	FUNCTION FC 817  : VOID
	TITLE =MAL1S017 Section control: LINE 1 SEC 17 GERM 1
	//COPYRIGHT:    (C) 2009 BY  BUHLER AG
	//                           CH-9240 UZWIL  SWITZERLAND
	//
	//PRODUCT:      WinCoS_BIW01_09
	//
	//TITLE:        LINE 1 SEC 17 GERM 1
	//                 Section control
	//
	//--------------------------------------------------------------------------------
	//
	//IDENT:        AUTHOR:             DEPT:                              DATE:
	//
	//P01_FC817.1.0 K.Renz              CSB41                              13.Jan.2010
	//              1st Release
	//
	//--------------------------------------------------------------------------------
	//
	//PURPOSE:
	//
	//REFERENCES : GCSOSMAN
	//
	//--------------------------------------------------------------------------------
	//
	//
	AUTHOR  : KR
	FAMILY  : USW
	VERSION : 9.9
	//0000 to 0999: Main Functions
	//              0 =Main Function Cylic
	//              1 =Main Function Coldstart/Newstart
	//              2 =Main Function Warm Start

	VAR_INPUT
	  InCode : INT ;
	END_VAR

	VAR_TEMP
	tmpStartNext : BOOL ;	//Condition to Start next element
	tmpFlagFault : BOOL ;	//Flag mechanical fault
	tmpEnableFeed : BOOL ;
	tmpStartScale : BOOL ;
	tmpStartLiqScale : BOOL ; //Enable to Start Lipquid Scale
	tmpSndBin: Int ;
	tmpRcvBin: Int ;
	tmpBool : BOOL ;
	tmpByte : BYTE ;
	tmpWord : WORD ;
	tmpDWord : DWORD ;
	tmpInt : INT ;
	tmpRET : INT ;
	tmpDInt : DINT ;
	tmpCyclusTime : DINT ;
	tmpWetSteep : BOOL ;
	END_VAR

	BEGIN

	NETWORK
	TITLE =
	//=================================================
	//=================================================
	//S T A R T   M A I N   F U N C T I O N
	//=================================================
	//=================================================
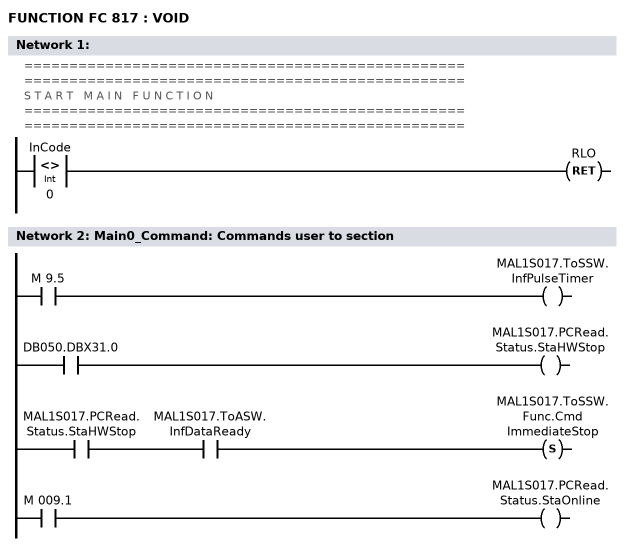
	      L InCode;
	      L 0;
	      <>I;
	      BEB;

	NETWORK
	TITLE =Main0_Command: Commands user to section
	      NOP   0;
	//-Tick 1 second---
		U     M 9.5;
		=     MAL1S017.ToSSW.InfPulseTimer;
	//-Hardware stop---
		U     DB050.DBX31.0 ;
		=     MAL1S017.PCRead.Status.StaHWStop;
		U   MAL1S017.PCRead.Status.StaHWStop;
		U   MAL1S017.ToASW.InfDataReady;
		S     MAL1S017.ToSSW.Func.CmdImmediateStop;
	//-Online---
		U     M 009.1 ;
		=     MAL1S017.PCRead.Status.StaOnline;
	NETWORK
	TITLE =ASW_UC: User commands to section
	NOP 0;
	//-Additional user commands---
	//-GP standard commands---
	      AUF   "MAL1S017" ;
	      L     L#0 ;                           // Enter the differenz of the target weight and prestop weight
	      T    "MAL1S017".VarTemp.InOutValue3;  // Prestop weight
	      CALL FC   120 (
	           InCode                   := 2001);// Section function: Standard section commands

	//-Condition CmdSequenzStop---
	      U     MAL1S017.ToSSW.Func.CmdSequenzStop;
	//      S     "MAL1S017".ToSSW.Func.CmdSequenzStop
	      R     MAL1S017.ToSSW.Func.CmdSequenzStop;
	//-Extended section commands---
	      AUF   "MAL1S017";
	      CALL "STD_LineSecStdSub" (
	           InCode                   := 2002);// Section function: Extended section commands
	//-Status from pulse commands---
	      CLR;
	      =     DB817.DBX  157.0;
	      =     DB817.DBX  157.1;
	      =     DB817.DBX  157.2;
	      =     DB817.DBX  157.3;
	      =     DB817.DBX  157.4;
	      =     DB817.DBX  157.5;
	      =     DB817.DBX  157.6;
	      =     DB817.DBX  157.7;
	//
	NETWORK
	TITLE =Main0_Dest: Destination
	NETWORK
	TITLE =Main0_Next: Ready for next batch

		ON    MAL1S017.ToASW.InfDataReady;
		=     MAL1S017.ToSSW.InfReadyForNewBatch;
	NETWORK
	TITLE =Main0_Control: Control section
	      NOP   0;
	//-Process commands from PCS---
		AUF   "MAL1S017" ;
		CALL FC    60 (// Methode O_Section
		CODE                     := 7);
	//-Process commands from user---
		AUF   "MAL1S017" ;
		CALL FC    60 (// Methode Control
		CODE                     := 0);
	//-Process section step---
		AUF   "MAL1S017" ;
		CALL FC    60 (// Methode Step_execute
		CODE                     := 2);
		AUF   "MAL1S017" ;
		CALL FC    60 (// Methode Step_transition
		CODE                     := 3);
	//-Process section state---
		AUF   "MAL1S017" ;
		CALL FC    60 (// Methode State
		CODE                     := 4);

	NETWORK
	TITLE =Main0_Init: Init
		UN    MAL1S017.ToASW.Transition.ToWait;
		UN    MAL1S017.ToASW.CmdNewBatch;
		SPB   in00;
	//-User initialization---
		AUF   "MAL1S017" ;
	//
	//-Section function: Init ---
		AUF   "MAL1S017" ;
	      CALL FC   120 (
	           InCode                   := 2003);// Section function: Init
	//
	//-Group interface---
	//
	//-Initialise bin objects---
	//
	//-Emptying job---
	      U    MAL1S017.JobAc.StaBatch.StaEmptyingBatch;
	      S     MAL1S017.PCRead.Status.StaLoaded;
	//
	//-Error Batch---
	//
	in00:	NOP   0;

	NETWORK
	TITLE =ASW_VB: Various functions before bin control
	      NOP   0;
	//
	//-Update staSameSndRcv in sender binlist---
	NETWORK
	TITLE =Main0_GrNRS: Not Relevant for started / Fault
		NOP 0;
	      SET;
	      =     "MAL1S017".Gr.ParNotRelForStarted[103];
	      =     "MAL1S017".Gr.ParNotRelForStarted[105];
	      =     "MAL1S017".Gr.ParNotRelForStarted[106];
	      =     "MAL1S017".Gr.ParNotRelForStarted[107];
	      =     "MAL1S017".Gr.ParNotRelForStarted[108];
	      =     "MAL1S017".Gr.ParNotRelForStarted[109];
	      =     "MAL1S017".Gr.ParNotRelForStarted[112];
	      =     "MAL1S017".Gr.ParNotRelForFault[103];
	      =     "MAL1S017".Gr.ParNotRelForFault[105];
	      =     "MAL1S017".Gr.ParNotRelForFault[106];
	      =     "MAL1S017".Gr.ParNotRelForFault[107];
	      =     "MAL1S017".Gr.ParNotRelForFault[108];
	      =     "MAL1S017".Gr.ParNotRelForFault[109];
	      =     "MAL1S017".Gr.ParNotRelForFault[112];
	NETWORK
	TITLE =Main0_GrSelection: Group selection
	// List of the used objects in the section
	// ==========================
	// G005G       GENERAL ELEMENTS GERM 1
	// G091F       BELT CONVEYOR 4100 GERM 1-4
	// G092F       BELT CONVEYOR 4200 GERM 5-8
	// G093M       BELT CONVEYOR 4300 GERM
	// G094M       BELT CONVEYOR 4400 GERM
	// G095M       BELT CONVEYOR 4500 GERM
	// G097M       LIFTING DEVICE GERM 1
	// G098M       COUPLING DEVICE TURNER GERM 1
	// G099M       COUPLING DEVICE WALL GERM 1
	// G100M       TRAVELLING DRIVE GERM 1
	// G101M       HORIZONTAL AND LIFTING SCREW GERM 1
	// G102M       LOCAL COMMAND BUTTON / LAMPS GERM 1
	// G103M       TEMPERATURE MES. GERM 1
	// G104M       TURNING SCREWS GERM 1
	// G105M       FAN AND VALVE SRAY AIR GERM 1
	// G106M       FRESH AIR LOUVER GERM 1
	// G107M       EXHAUST AIR LOUVER GERM 1
	// G108M       PRODUCT MOISTERING  GERM 1
	// G109M       HP CLEANING GERM 1
	// G110M       INLET SLIDE GERM 1
	// G111M       LOADING CONVEYOR 4600 GERM 1
	// G112M       COOLING / HEATING GERM 1
	// G113M       BELT CONVEYOR 7050 GERM 1 / 2
	//
	      NOP   0;
//-Condition for preselection---
		U     MAL1S017.ToASW.InfDataReady;
		SPB   GS01;
//-Deselect groups ---
		CALL FB     9 , "GCS7_GrCtrlDBTmp" (// GrCtr.Methode Deselect
		     Code  := 3,
		     Sec   := "MAL1S017".Gr);
		SPA   GS02;
//-Select groups ---
	GS01:	NOP 0;
	//-Prepare for preselection ---
		CALL FB     9 , "GCS7_GrCtrlDBTmp" (// GrCtr.Methode Init Preselection
		     Code  := 1,
		     Sec   := "MAL1S017".Gr);
	//
	//
	//-Prestart used groups --
		U     M     50.0;
		=     M     50.0;

	//-Preselect used groups --
		U     M     50.0;
		=     M     50.0;
		S   MAL1S017.Gr.InPreselect[5];   //-->G005G GENERAL ELEMENTS GERM 1
		S   MAL1S017.Gr.InPreselect[91];   //-->G091F BELT CONVEYOR 4100 GERM 1-4
		S   MAL1S017.Gr.InPreselect[92];   //-->G092F BELT CONVEYOR 4200 GERM 5-8
		S   MAL1S017.Gr.InPreselect[93];   //-->G093M BELT CONVEYOR 4300 GERM
		S   MAL1S017.Gr.InPreselect[94];   //-->G094M BELT CONVEYOR 4400 GERM
		S   MAL1S017.Gr.InPreselect[95];   //-->G095M BELT CONVEYOR 4500 GERM
		S   MAL1S017.Gr.InPreselect[97];   //-->G097M LIFTING DEVICE GERM 1
		S   MAL1S017.Gr.InPreselect[98];   //-->G098M COUPLING DEVICE TURNER GERM 1
		S   MAL1S017.Gr.InPreselect[99];   //-->G099M COUPLING DEVICE WALL GERM 1
		S   MAL1S017.Gr.InPreselect[100];   //-->G100M TRAVELLING DRIVE GERM 1
		S   MAL1S017.Gr.InPreselect[101];   //-->G101M HORIZONTAL AND LIFTING SCREW GERM 1
		S   MAL1S017.Gr.InPreselect[102];   //-->G102M LOCAL COMMAND BUTTON / LAMPS GERM 1
		S   MAL1S017.Gr.InPreselect[103];   //-->G103M TEMPERATURE MES. GERM 1
		S   MAL1S017.Gr.InPreselect[104];   //-->G104M TURNING SCREWS GERM 1
		S   MAL1S017.Gr.InPreselect[105];   //-->G105M FAN AND VALVE SRAY AIR GERM 1
		S   MAL1S017.Gr.InPreselect[106];   //-->G106M FRESH AIR LOUVER GERM 1
		S   MAL1S017.Gr.InPreselect[107];   //-->G107M EXHAUST AIR LOUVER GERM 1
		S   MAL1S017.Gr.InPreselect[108];   //-->G108M PRODUCT MOISTERING  GERM 1
		S   MAL1S017.Gr.InPreselect[109];   //-->G109M HP CLEANING GERM 1
		S   MAL1S017.Gr.InPreselect[110];   //-->G110M INLET SLIDE GERM 1
		S   MAL1S017.Gr.InPreselect[111];   //-->G111M LOADING CONVEYOR 4600 GERM 1
		S   MAL1S017.Gr.InPreselect[112];   //-->G112M COOLING / HEATING GERM 1
		S   MAL1S017.Gr.InPreselect[113];   //-->G113M BELT CONVEYOR 7050 GERM 1 / 2
	      L     1;
	      L     "MAL1S017Par".StepAct.StepNumber;
	      UW;
	      ==I;  // step wetsteep
	      =    "MAL1S017Par".Par.FlagGen.WetStep;

	//
	//-Set CmdNewJob ---
	     U     MAL1S017.Gr.InPreselect[91];
	     UN    #GCS7_GrCtrlDB.OutOccupied[91];
	     S       G091F.CmdNewJob;
	     U     MAL1S017.Gr.InPreselect[92];
	     UN    #GCS7_GrCtrlDB.OutOccupied[92];
	     S       G092F.CmdNewJob;
	     U     MAL1S017.Gr.InPreselect[93];
	     UN    #GCS7_GrCtrlDB.OutOccupied[93];
	     S       G093M.CmdNewJob;
	     U     MAL1S017.Gr.InPreselect[94];
	     UN    #GCS7_GrCtrlDB.OutOccupied[94];
	     S       G094M.CmdNewJob;
	     U     MAL1S017.Gr.InPreselect[95];
	     UN    #GCS7_GrCtrlDB.OutOccupied[95];
	     S       G095M.CmdNewJob;
	     U     MAL1S017.Gr.InPreselect[97];
	     UN    #GCS7_GrCtrlDB.OutOccupied[97];
	     S       G097M.CmdNewJob;
	     U     MAL1S017.Gr.InPreselect[98];
	     UN    #GCS7_GrCtrlDB.OutOccupied[98];
	     S       G098M.CmdNewJob;
	     U     MAL1S017.Gr.InPreselect[99];
	     UN    #GCS7_GrCtrlDB.OutOccupied[99];
	     S       G099M.CmdNewJob;
	     U     MAL1S017.Gr.InPreselect[100];
	     UN    #GCS7_GrCtrlDB.OutOccupied[100];
	     S       G100M.CmdNewJob;
	     U     MAL1S017.Gr.InPreselect[101];
	     UN    #GCS7_GrCtrlDB.OutOccupied[101];
	     S       G101M.CmdNewJob;
	     U     MAL1S017.Gr.InPreselect[102];
	     UN    #GCS7_GrCtrlDB.OutOccupied[102];
	     S       G102M.CmdNewJob;
	     U     MAL1S017.Gr.InPreselect[103];
	     UN    #GCS7_GrCtrlDB.OutOccupied[103];
	     S       G103M.CmdNewJob;
	     U     MAL1S017.Gr.InPreselect[104];
	     UN    #GCS7_GrCtrlDB.OutOccupied[104];
	     S       G104M.CmdNewJob;
	     U     MAL1S017.Gr.InPreselect[105];
	     UN    #GCS7_GrCtrlDB.OutOccupied[105];
	     S       G105M.CmdNewJob;
	     U     MAL1S017.Gr.InPreselect[106];
	     UN    #GCS7_GrCtrlDB.OutOccupied[106];
	     S       G106M.CmdNewJob;
	     U     MAL1S017.Gr.InPreselect[107];
	     UN    #GCS7_GrCtrlDB.OutOccupied[107];
	     S       G107M.CmdNewJob;
	     U     MAL1S017.Gr.InPreselect[108];
	     UN    #GCS7_GrCtrlDB.OutOccupied[108];
	     S       G108M.CmdNewJob;
	     U     MAL1S017.Gr.InPreselect[109];
	     UN    #GCS7_GrCtrlDB.OutOccupied[109];
	     S       G109M.CmdNewJob;
	     U     MAL1S017.Gr.InPreselect[110];
	     UN    #GCS7_GrCtrlDB.OutOccupied[110];
	     S       G110M.CmdNewJob;
	     U     MAL1S017.Gr.InPreselect[111];
	     UN    #GCS7_GrCtrlDB.OutOccupied[111];
	     S       G111M.CmdNewJob;
	     U     MAL1S017.Gr.InPreselect[112];
	     UN    #GCS7_GrCtrlDB.OutOccupied[112];
	     S       G112M.CmdNewJob;
	     U     MAL1S017.Gr.InPreselect[113];
	     UN    #GCS7_GrCtrlDB.OutOccupied[113];
	     S       G113M.CmdNewJob;
	//
	//
	//-Test preselected groups ---
		CALL FB     9 , "GCS7_GrCtrlDBTmp" (// GrCtr.Methode Select
		     Code  := 2,
		     Sec   := "MAL1S017".Gr);
	//
	//-Way conflict if not available---
		CLR;
		S     MAL1S017.Gr.All.OutGrConflict;
	//
	//-Test occupied real and virtual groups---
	GS02:   NOP 0;
		U     MAL1S017.Gr.All.OutSelectionValid;
		UN    MAL1S017.Gr.All.OutGrIsLocked;
		=     MAL1S017.Gr.All.InOutASWSelectionOK;
	//
	//
	//----- Send data to selected groups =====
	GS3:	UN  MAL1S017.Gr.OutSelected[91]; //G091F
		SPB GS4;
		L     "MAL1".Para.ParLineNr;
		T     G091F.Gr.InLine;
	GS4:	UN  MAL1S017.Gr.OutSelected[92]; //G092F
		SPB GS5;
		L     "MAL1".Para.ParLineNr;
		T     G092F.Gr.InLine;
	GS5:	UN  MAL1S017.Gr.OutSelected[93]; //G093M
		SPB GS6;
		L     "MAL1".Para.ParLineNr;
		T     G093M.Gr.InLine;
	GS6:	UN  MAL1S017.Gr.OutSelected[94]; //G094M
		SPB GS7;
		L     "MAL1".Para.ParLineNr;
		T     G094M.Gr.InLine;
	GS7:	UN  MAL1S017.Gr.OutSelected[95]; //G095M
		SPB GS8;
		L     "MAL1".Para.ParLineNr;
		T     G095M.Gr.InLine;
	GS8:	UN  MAL1S017.Gr.OutSelected[97]; //G097M
		SPB GS9;
		L     "MAL1".Para.ParLineNr;
		T     G097M.Gr.InLine;
	GS9:	UN  MAL1S017.Gr.OutSelected[98]; //G098M
		SPB GS10;
		L     "MAL1".Para.ParLineNr;
		T     G098M.Gr.InLine;
	GS10:	UN  MAL1S017.Gr.OutSelected[99]; //G099M
		SPB GS11;
		L     "MAL1".Para.ParLineNr;
		T     G099M.Gr.InLine;
	GS11:	UN  MAL1S017.Gr.OutSelected[100]; //G100M
		SPB GS12;
		L     "MAL1".Para.ParLineNr;
		T     G100M.Gr.InLine;
	GS12:	UN  MAL1S017.Gr.OutSelected[101]; //G101M
		SPB GS13;
		L     "MAL1".Para.ParLineNr;
		T     G101M.Gr.InLine;
	GS13:	UN  MAL1S017.Gr.OutSelected[102]; //G102M
		SPB GS14;
		L     "MAL1".Para.ParLineNr;
		T     G102M.Gr.InLine;
	GS14:	UN  MAL1S017.Gr.OutSelected[103]; //G103M
		SPB GS15;
		L     "MAL1".Para.ParLineNr;
		T     G103M.Gr.InLine;
	GS15:	UN  MAL1S017.Gr.OutSelected[104]; //G104M
		SPB GS16;
		L     "MAL1".Para.ParLineNr;
		T     G104M.Gr.InLine;
	GS16:	UN  MAL1S017.Gr.OutSelected[105]; //G105M
		SPB GS17;
		L     "MAL1".Para.ParLineNr;
		T     G105M.Gr.InLine;
	GS17:	UN  MAL1S017.Gr.OutSelected[106]; //G106M
		SPB GS18;
		L     "MAL1".Para.ParLineNr;
		T     G106M.Gr.InLine;
	GS18:	UN  MAL1S017.Gr.OutSelected[107]; //G107M
		SPB GS19;
		L     "MAL1".Para.ParLineNr;
		T     G107M.Gr.InLine;
	GS19:	UN  MAL1S017.Gr.OutSelected[108]; //G108M
		SPB GS20;
		L     "MAL1".Para.ParLineNr;
		T     G108M.Gr.InLine;
	GS20:	UN  MAL1S017.Gr.OutSelected[109]; //G109M
		SPB GS21;
		L     "MAL1".Para.ParLineNr;
		T     G109M.Gr.InLine;
	GS21:	UN  MAL1S017.Gr.OutSelected[110]; //G110M
		SPB GS22;
		L     "MAL1".Para.ParLineNr;
		T     G110M.Gr.InLine;
	GS22:	UN  MAL1S017.Gr.OutSelected[111]; //G111M
		SPB GS23;
		L     "MAL1".Para.ParLineNr;
		T     G111M.Gr.InLine;
	GS23:	UN  MAL1S017.Gr.OutSelected[112]; //G112M
		SPB GS24;
		L     "MAL1".Para.ParLineNr;
		T     G112M.Gr.InLine;
	GS24:	UN  MAL1S017.Gr.OutSelected[113]; //G113M
		SPB GS25;
		L     "MAL1".Para.ParLineNr;
		T     G113M.Gr.InLine;
	GS25:	NOP 0;
	NETWORK
	TITLE =Main0_GrCmd: CMD section to Groups

		NOP   0;
//-Way Adjust Time---
		O     MAL1S017.Gr.All.CmdNewSelection;
		O     MAL1S017.ToASW.CmdModify;
		S     MAL1S017.ToSSW.CmdNewWay;
		AUF   "MAL1S017" ;
		CALL FC    60 (// Methode Adjust Time
		CODE                     := 13);
//-Continue---
		U     MAL1S017.ToASW.Func.CmdStart;
		O     MAL1S017.ToASW.Func.CmdNextStep;
		S     MAL1S017.Gr.All.CmdContinue;
//-Fault reset---
		U     MAL1S017.ToASW.Func.CmdFaultReset;
		S     MAL1S017.Gr.All.CmdFaultReset;
//-Manual mode---
		U     MAL1S017.ToASW.Func.CmdAutomatic;
		S     MAL1S017.Gr.All.CmdManualOff;
		UN     MAL1S017.PCRead.Status.StaHand;
		S     MAL1S017.Gr.All.CmdManualOffRel;
//-Clear idling---
		U     MAL1S017.PCRead.Status.StaImmediateStopASW;
		S     MAL1S017.Gr.All.CmdClearIdling;
//-Start next---
		UN    MAL1S017.PCRead.Status.StaStep;
		O     MAL1S017.ToASW.Func.CmdNextStep;
		U(;
		L       MAL1S017.PCRead.OutWayAdjustTime;
		L     2;
		>I;
		O     MAL1S017.ToASW.InfWayAdjustTimeEnd;
		);
		UN    MAL1S017.Gr.All.CmdNewSelection;
		UN    MAL1S017.PCRead.Step.StWait;
		=     #tmpStartNext; //-->VarStartNext
//-Start next feed---
		U     MAL1S017.Gr.Wgr.OutStartedRel;
		ON    MAL1S017.ToASW.InfWayAdjustTimeEnd;
		UN    MAL1S017.PCRead.Status.StaFeedOffASW;
		UN    MAL1S017.PCRead.Status.StaImmediateStopASW;
		U     MAL1S017.Gr.Mgr.OutStartedRel;
		U     MAL1S017.PCRead.Step.StActive;
		=     MAL1S017.Gr.Feed.InEnable;
		=     #tmpEnableFeed;
		U     #tmpStartNext;
		U     MAL1S017.Gr.Wgr.OutStartedRel;
		U     MAL1S017.Gr.All.OutAutoStartOk;
		U     MAL1S017.PCRead.Status.StaAutostartSec;
		=     MAL1S017.Gr.Feed.CmdNext;
//-Start next machine group---
		UN    MAL1S017.PCRead.Status.StaImmediateStopASW;
		=     MAL1S017.Gr.Mgr.InEnable;
		U     #tmpStartNext;
		=     MAL1S017.Gr.Mgr.CmdNext;
//-Start next way group---
		UN    MAL1S017.PCRead.Status.StaImmediateStopASW;
		=     MAL1S017.Gr.Wgr.InEnable;
		UN    MAL1S017.PCRead.Status.StaStep;
		O     MAL1S017.ToASW.Func.CmdNextStep;
		=     MAL1S017.Gr.Wgr.CmdNext;
//-Start next general group---
		UN    MAL1S017.PCRead.Status.StaImmediateStopASW;
		=     MAL1S017.Gr.Ggr.InEnable;
		U     #tmpStartNext;
		=     MAL1S017.Gr.Ggr.CmdNext;
//-Update command state---
		CALL FB     9 , "GCS7_GrCtrlDBTmp" (// GrCtr.Methode UpdateCmdSt
		     Code  := 4,
		     Sec   := "MAL1S017".Gr);

	NETWORK
	TITLE =Main0_Status: Fault/Status

		NOP   0;
//- Autostart Section---
		UN    MAL1S017.ToASW.Func.CmdStart;
		O     MAL1S017.Gr.All.OutAutoStartOk;
		=     MAL1S017.TimeoutAutostart.EN;
		CALL FC18 (
		   IN                       := MAL1S017.TimeoutAutostart.EN,
		   PT                       := 10,
		   Q                        := MAL1S017.TimeoutAutostart.Q,
		ET                       := MAL1S017.TimeoutAutostart.ET);
		U     MAL1S017.TimeoutAutostart.Q;
		UN     MAL1S017.Gr.All.OutAutoStartOk;
		R     MAL1S017.PCRead.Status.StaAutostartSec;
		U     MAL1S017.ToASW.Func.CmdStart;
		ON    MAL1S017.ToASW.InfDataReady;
		S     MAL1S017.PCRead.Status.StaAutostartSec;
//-Stopped---
		UN    MAL1S017.Gr.Mgr.InEnable;
		U     MAL1S017.Gr.All.OutStoppedRel;
		O     MAL1S017.Gr.All.OutStoppedAll;
		UN    MAL1S017.PCRead.Status.StaStep;
		O;
		U     MAL1S017.Gr.Mgr.OutStoppedRel;
		U     MAL1S017.PCRead.Status.StaStep;
		=     MAL1S017.ToSSW.InfStopped;
//-Started---
		U     MAL1S017.Gr.Mgr.OutStartedRel;
		=     MAL1S017.ToSSW.InfStarted;
//-Feeding---
		U     MAL1S017.Gr.Feed.InEnable; //Section without Feed groups
		ON    MAL1S017.Gr.Feed.OutStoppedAll;
		U     MAL1S017.Gr.Feed.OutStartedRel;
		=     MAL1S017.ToSSW.InfFeeding;
//-Autostart---
		U     MAL1S017.Gr.All.OutAutostartOkAll;
		U     MAL1S017.PCRead.Status.StaAutostartSec;
		=     MAL1S017.PCRead.Status.StaAutostart;
//-DPFault---
		U     MAL1S017.Gr.All.OutDPFault;
		=     MAL1S017.PCRead.Status.StaDPFault;
		S       MAL1S017.ToSSW.Func.CmdFeedOff;
//-Startwarning---
		U     MAL1S017.Gr.All.OutStartWarning;
		=     MAL1S017.PCRead.Status.StaStartwarning;
//-Way conflict---
		U     MAL1S017.Gr.All.OutGrConflict;
		=     MAL1S017.PCRead.Fault.EsWayConflict;
//-Warning---
		U     MAL1S017.Gr.All.OutWarning;
		=     MAL1S017.PCRead.Fault.EsWarning;
//-Fault---
		U     MAL1S017.Gr.All.OutFaultRel;
		FP      MAL1S017.PCRead.Fault.EsMech;
		S       MAL1S017.ToSSW.Func.CmdFeedOff;
//-Sender empty---
		CLR;
		=     MAL1S017.PCRead.Fault.EsEmpty; //-->Sec.EsEmpty
//-Receiver full---
		CLR;
		=     MAL1S017.PCRead.Fault.EsFull;

	NETWORK
	TITLE =Main0_StatusASW: Status from ASW
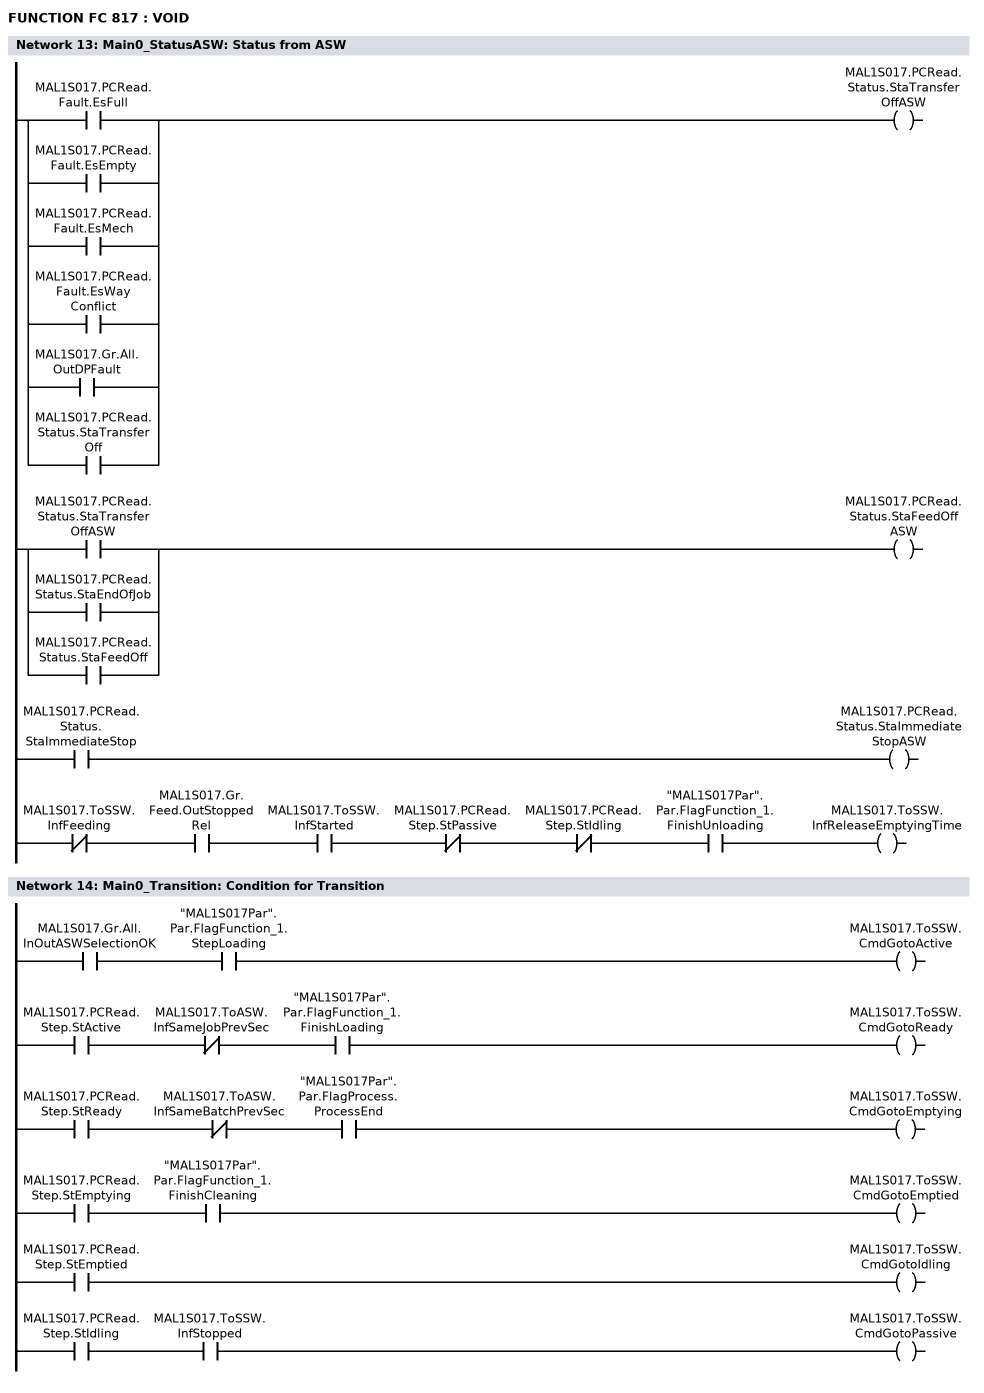
		NOP   0;
//-Transfer off with automatic restart---
		O     MAL1S017.PCRead.Fault.EsFull;
		O     MAL1S017.PCRead.Fault.EsEmpty;
		O     MAL1S017.PCRead.Fault.EsMech;
		O     MAL1S017.PCRead.Fault.EsWayConflict;
		O     MAL1S017.Gr.All.OutDPFault;
		O     MAL1S017.PCRead.Status.StaTransferOff;
		=     MAL1S017.PCRead.Status.StaTransferOffASW;
//-Feed off with automatic restart---
		U     MAL1S017.PCRead.Status.StaTransferOffASW;
		O     MAL1S017.PCRead.Status.StaEndOfJob; //
		O     MAL1S017.PCRead.Status.StaFeedOff;
		=     MAL1S017.PCRead.Status.StaFeedOffASW;
//-Immediate stop with automatic restart---
		U     MAL1S017.PCRead.Status.StaImmediateStop;
		=     MAL1S017.PCRead.Status.StaImmediateStopASW;
//-Emptying time---
	      UN   MAL1S017.ToSSW.InfFeeding;
	      U     MAL1S017.Gr.Feed.OutStoppedRel;
	      U     MAL1S017.ToSSW.InfStarted;
	      UN  MAL1S017.PCRead.Step.StPassive;
	      UN  MAL1S017.PCRead.Step.StIdling;
		U     "MAL1S017Par".Par.FlagFunction_1.FinishUnloading;
		=     MAL1S017.ToSSW.InfReleaseEmptyingTime;
	NETWORK
	TITLE =Main0_Transition: Condition for Transition

		NOP 0;
		NOP 0;
	//-Active---
		U   MAL1S017.Gr.All.InOutASWSelectionOK;
		U     "MAL1S017Par".Par.FlagFunction_1.StepLoading;
		=     MAL1S017.ToSSW.CmdGotoActive;
	//-Ready---
	        U    MAL1S017.PCRead.Step.StActive;
		UN   MAL1S017.ToASW.InfSameJobPrevSec;
		U     "MAL1S017Par".Par.FlagFunction_1.FinishLoading;
		=     MAL1S017.ToSSW.CmdGotoReady;
	//-Emptying---
	        U    MAL1S017.PCRead.Step.StReady;
		UN   MAL1S017.ToASW.InfSameBatchPrevSec;
		U     "MAL1S017Par".Par.FlagProcess.ProcessEnd;
		=     MAL1S017.ToSSW.CmdGotoEmptying;
	//-Emptied---
	        U    MAL1S017.PCRead.Step.StEmptying;
		U     "MAL1S017Par".Par.FlagFunction_1.FinishCleaning;
		=     MAL1S017.ToSSW.CmdGotoEmptied;
	//-Result section---
	//-Idling---
		U     MAL1S017.PCRead.Step.StEmptied;
		=     MAL1S017.ToSSW.CmdGotoIdling;
	//-Passive---
		U     MAL1S017.PCRead.Step.StIdling;
		U     MAL1S017.ToSSW.InfStopped;
		=     MAL1S017.ToSSW.CmdGotoPassive;
	NETWORK
	TITLE =Main0_Move: Move to next section
		NOP 0;
//-------------------------------------------
//-General Condition for move
//-------------------------------------------
		U   MAL1S017.PCRead.Step.StReady;
		SPBN  Move;
	//->Move batch to section MAL1S018
		AUF   "MAL1S017" ;
		CALL FC    60 (// Methode Move Data
		  CODE                     := 5);
		UN  MAL1S017.ToASW.CmdDataMoved;
		SPB Move;
	Move:	NOP 0;
	NETWORK
	TITLE =ASW_AH:Alarm horns
	      UN    MAL1S017.ToASW.Func.CmdHornOn;
	      SPB   AHJ1;
	      CALL "SYS_Horn_Code" (
	           FcCode                   := 1, //Set Alarm
	           ParObjectType            := 4000,
	           ParObjectNo              := 0,
	           ParHornCode              := 98);
	AHJ1: UN    MAL1S017.ToASW.Func.CmdHornOff;
	      SPB   AH00;
	      CALL "SYS_Horn_Code" (
	           FcCode                   := 2, //Reset Alarm
	           ParObjectType            := 4000,
	           ParObjectNo              := 0,
	           ParHornCode              := 1);
	      CALL "SYS_Horn_Code" (
	           FcCode                   := 2, //Reset Alarm
	           ParObjectType            := 4000,
	           ParObjectNo              := 0,
	           ParHornCode              := 2);
	      CALL "SYS_Horn_Code" (
	           FcCode                   := 2, //Reset Alarm
	           ParObjectType            := 4000,
	           ParObjectNo              := 0,
	           ParHornCode              := 99);
	AH00: NOP   0;
	NETWORK
	TITLE =ASW_FT: Feeding Time
		AUF   "MAL1S017" ;
	      CALL FC   120 (
	           InCode                 := 2004);// Section function: Feeding time

	NETWORK
	TITLE =ASW_OL: Override low level
	//
		AUF   "MAL1S017" ;
	//
	OL00: NOP   0;
	NETWORK
	TITLE =ASW_VA: VA Various functions after section control
	//
		AUF   "MAL1S017" ;
	// Copy bin number to section DB
	        L   MAL1S017.JobAc.BatchSndBin;
		L   MAL1S017.MAL1S001SND33.Ingr[1].Bin;
	        T   MAL1S017.JobAc.BatchSndBin;
		<>I;
		S   MAL1S017.ChangeBit.CBit1;
		//
	        L   MAL1S017.JobAc.BatchRcvBin;
		L   MAL1S017.MAL1S001RCV34.Ingr[1].Bin;
	        T   MAL1S017.JobAc.BatchRcvBin;
		<>I;
		S   MAL1S017.ChangeBit.CBit1;
		//
	        L   MAL1S017.JobAc.BatchRcvBin;
		L   MAL1S017.MAl1S034RCV36.Ingr[1].Bin;
	        T   MAL1S017.JobAc.BatchRcvBin;
		<>I;
		S   MAL1S017.ChangeBit.CBit1;
		//

	NETWORK
	TITLE =ASW_EJ End of job
	NOP 0;
	//
	//-Fluidlift monitoring---
	NETWORK
	TITLE =ASW_VE: VE New value event
	//
	//-Group interface---
	      U    MAL1S017.ToASW.CmdModify;
	      S     G091F.CmdNewValue;
	      S     G092F.CmdNewValue;
	      S     G093M.CmdNewValue;
	      S     G094M.CmdNewValue;
	      S     G095M.CmdNewValue;
	      S     G097M.CmdNewValue;
	      S     G098M.CmdNewValue;
	      S     G099M.CmdNewValue;
	      S     G100M.CmdNewValue;
	      S     G101M.CmdNewValue;
	      S     G102M.CmdNewValue;
	      S     G103M.CmdNewValue;
	      S     G104M.CmdNewValue;
	      S     G105M.CmdNewValue;
	      S     G106M.CmdNewValue;
	      S     G107M.CmdNewValue;
	      S     G108M.CmdNewValue;
	      S     G109M.CmdNewValue;
	      S     G110M.CmdNewValue;
	      S     G111M.CmdNewValue;
	      S     G112M.CmdNewValue;
	      S     G113M.CmdNewValue;


	NETWORK
	TITLE =ASW_NV: New value data
	NETWORK
	TITLE =ASW_WJ: Weight job
	//
	      U     MAL1S017.PCRead.Step.StActive;
	      O     MAL1S017.PCRead.Step.StReady;
	      O     MAL1S017.PCRead.Step.StEmptying;
	      O     MAL1S017.PCRead.Step.StEmptied;
	      SPBN   WJ08;
	//
	      L     MAL1S017.JobNom.JobWeight; //Target/Actual registration if no scale
	      T     MAL1S017.JobAc.JobWeight;
	//
	WJ08: NOP 0;
	//--------------------------------------------
	//PW Prestop weight
	//--------------------------------------------
	WJ00: NOP   0;
	NETWORK
	TITLE =ASW_SC: Section status text and colour
	//
		AUF   "MAL1S017" ;
	      CALL FC   120 (
	           InCode                   := 2055);// Section function: WinCoS.SectionInfoCode
	//
	NETWORK
	TITLE =ASW_5010: Prepare Log-Data cyclic
	// Prepare Log-Data cyclic
	      U     "MAL1S017".ToASW.InfDataReady; // job in section
	      U     M      4.7; // scan 30sec
	      SPBN  N501;
	      AUF   "MAL1S017";
	      L     0;
	      T     #tmpInt;
	      CALL "SIEMENS_FILL" (
		   BVAL                     := #tmpInt,
		   RET_VAL                  := #tmpRet,
		   BLK                      := "SSA_LOG_Value_Queue".Input);
	// header
	//
	      L     B#16#14; // type 20 = germinating
	      T     "SSA_LOG_Value_Queue".Input.Header.SecType; // type
	      L     B#16#1; // format 1 = cyclic
	      T     "SSA_LOG_Value_Queue".Input.Header.Format; // format
	      L     "MAL1S017".JobNom.JobNr;
	      T     "SSA_LOG_Value_Queue".Input.Para_0005;
	      L     "DB Prozesszeit".Sektion_17.Gesamtzeit_in_Minuten;
	      T     "SSA_LOG_Value_Queue".Input.Para_0007;
	      L     "MAL1S017Par".Par.ParIntMachine.ActualStep;
	      T     "SSA_LOG_Value_Queue".Input.Para_0008;
	      L     "MAL1S017Par".ActTimeStepProcess.SteptimeActMinOverall;
	      T     "SSA_LOG_Value_Queue".Input.Para_0009;
	//
	// values doubleword
	//=================================
	      L     G103M.A_2191_BTE02.OutValueUnits; // AIR TEMPERATURE ABOVE FLOOR
	      T     "SSA_LOG_Value_Queue".Input.Para_0015;
	//=================================
	      L     "MAL1S017Par".StepAct.TemperaturAboveFloor; // setpoint from SCADA
	      T     "SSA_LOG_Value_Queue".Input.Para_0017;
	//=================================
	      L     G103M.A_2191_BTE01.OutValueUnits; // AIR TEMPERATURE BELOW FLOOR
	      T     "SSA_LOG_Value_Queue".Input.Para_0019;
	//=================================
	      L     "MAL1S017Par".StepAct.TemperaturBelowFloor; // setpoint from SCADA
	      T     "SSA_LOG_Value_Queue".Input.Para_0021;
	//=================================
	      L     0; // Temperature low point of product
	      T     "SSA_LOG_Value_Queue".Input.Para_0023;
	//=================================
	      L     0; // Temperature middle point of product
	      T     "SSA_LOG_Value_Queue".Input.Para_0025;
	//=================================
	      L     0; // Temperature high point of product
	      T     "SSA_LOG_Value_Queue".Input.Para_0027;
	//=================================
	      L     0; // Temperature Spray Water
	      T     "SSA_LOG_Value_Queue".Input.Para_0029;
	//=================================
	      L     G106M.A_2151_MXZ01.OutPosition; // FRESH AIR FLAP 1
	      ITD;
	      T     "SSA_LOG_Value_Queue".Input.Para_0031;
	//=================================
	      L     0; // act position recycled air flap
	      T     "SSA_LOG_Value_Queue".Input.Para_0013;
	//=================================
	      L     G107M.A_2150_MXZ01.OutPosition; // LOUVER EXHAUST AIR
	      ITD;
	      T     "SSA_LOG_Value_Queue".Input.Para_0035;
	//=================================
	      L     0; // act position waste air flap 2
	      T     "SSA_LOG_Value_Queue".Input.Para_0037;
	//=================================
	      L     G105M.A_2160_TSC01_PD1.OutValueUnits; // FREQUENCY FREQ. GERM FAN 1
	      T     "SSA_LOG_Value_Queue".Input.Para_0039;
	//=================================
	      L     G105M.A_2160_TSC02_PD1.OutValueUnits; // FREQUENCY FREQ. GERM FAN 2
	      T     "SSA_LOG_Value_Queue".Input.Para_0041;
	//=================================
	      L     0; // spare
	      T     "SSA_LOG_Value_Queue".Input.Para_0043;
	//=================================
	      L     0; // spare
	      T     "SSA_LOG_Value_Queue".Input.Para_0045;
	//=================================
	      L     0; // spare
	      T     "SSA_LOG_Value_Queue".Input.Para_0047;
	//=================================
	      L     0; // spare
	      T     "SSA_LOG_Value_Queue".Input.Para_0049;
	//=================================
	      L     0; // spare
	      T     "SSA_LOG_Value_Queue".Input.Para_0051;
	// values integer bit info 0/1
	      L     L#0; // spare
	      T     "SSA_LOG_Value_Queue".Input.Para_0089;
	      L     L#0; // spare
	      T     "SSA_LOG_Value_Queue".Input.Para_0090;
	      L     L#0; // spare
	      T     "SSA_LOG_Value_Queue".Input.Para_0091;
	      L     L#0; // spare
	      T     "SSA_LOG_Value_Queue".Input.Para_0092;
	      U     "MAL1S017Par".Par.FlagProcess2.Turning1WithSpraying;
	      O     "MAL1S017Par".Par.FlagProcess2.Turning2WithSpraying;
	      L   1;
	      SPB MP93;
	      L   0;
	MP93: T     "SSA_LOG_Value_Queue".Input.Para_0093; // Spraying
	      U     "MAL1S017Par".Par.FlagFunction_1.StepCleaning; // Step Cleaning
	      L   1;
	      SPB MP94;
	      L   0;
	MP94: T     "SSA_LOG_Value_Queue".Input.Para_0094; // Cleaning
	      L   "MAL1S017Par".StepAct.Cooling;
	      L   1;
	      UW;
	MP95: T     "SSA_LOG_Value_Queue".Input.Para_0095; // Cooling

	      U     "MAL1S017Par".Par.FlagProcess2.Turning1WithoutSpraying;
	      O     "MAL1S017Par".Par.FlagProcess2.Turning2WithoutSpraying;
	      L   1;
	      SPB MP96;
	      L   0;
	MP96: T     "SSA_LOG_Value_Queue".Input.Para_0096; // Turning

	      U     M      9.0; // cooling on/off
	      L   1;
	      SPB MP97;
	      L   0;
	MP97: T     "SSA_LOG_Value_Queue".Input.Para_0097; // Spraying and Acid
	      L   "MAL1S017Par".StepAct.AirMoisten;
	      L   1;
	      UW;
	MP98: T     "SSA_LOG_Value_Queue".Input.Para_0098;  // Air Moisten

	//
	      NOP   0;
	// cont log-messages
	      L     "SSA_LOG_Value_Queue".Input.Para_0099; // message counter
	      L     1;
	      +I    ;
	      T     "SSA_LOG_Value_Queue".Input.Para_0099; // message counter

	// put timestamp into message
	      CALL "SIEMENS_BLKMOV" (
	           SRCBLK                   := "DB Prozesszeit".Arbeitsbereich.dt2,
	           RET_VAL                  := #tmpInt,
	           DSTBLK                   := "SSA_LOG_Value_Queue".Input.TimeStamp);
	//
	      CALL "SSA_MH_LogEntry_ActValue" (
	           DBNumber                 := 1005);
	N501: NOP   0;
	NETWORK
	TITLE =ASW_5020 :: Count electrical energy consumption
	//
	NETWORK
	TITLE =ASW_5030: Prepare Log-Data step values
	NOP 0;
	NETWORK
	TITLE =ASW_5060: Prepare Log-Data events
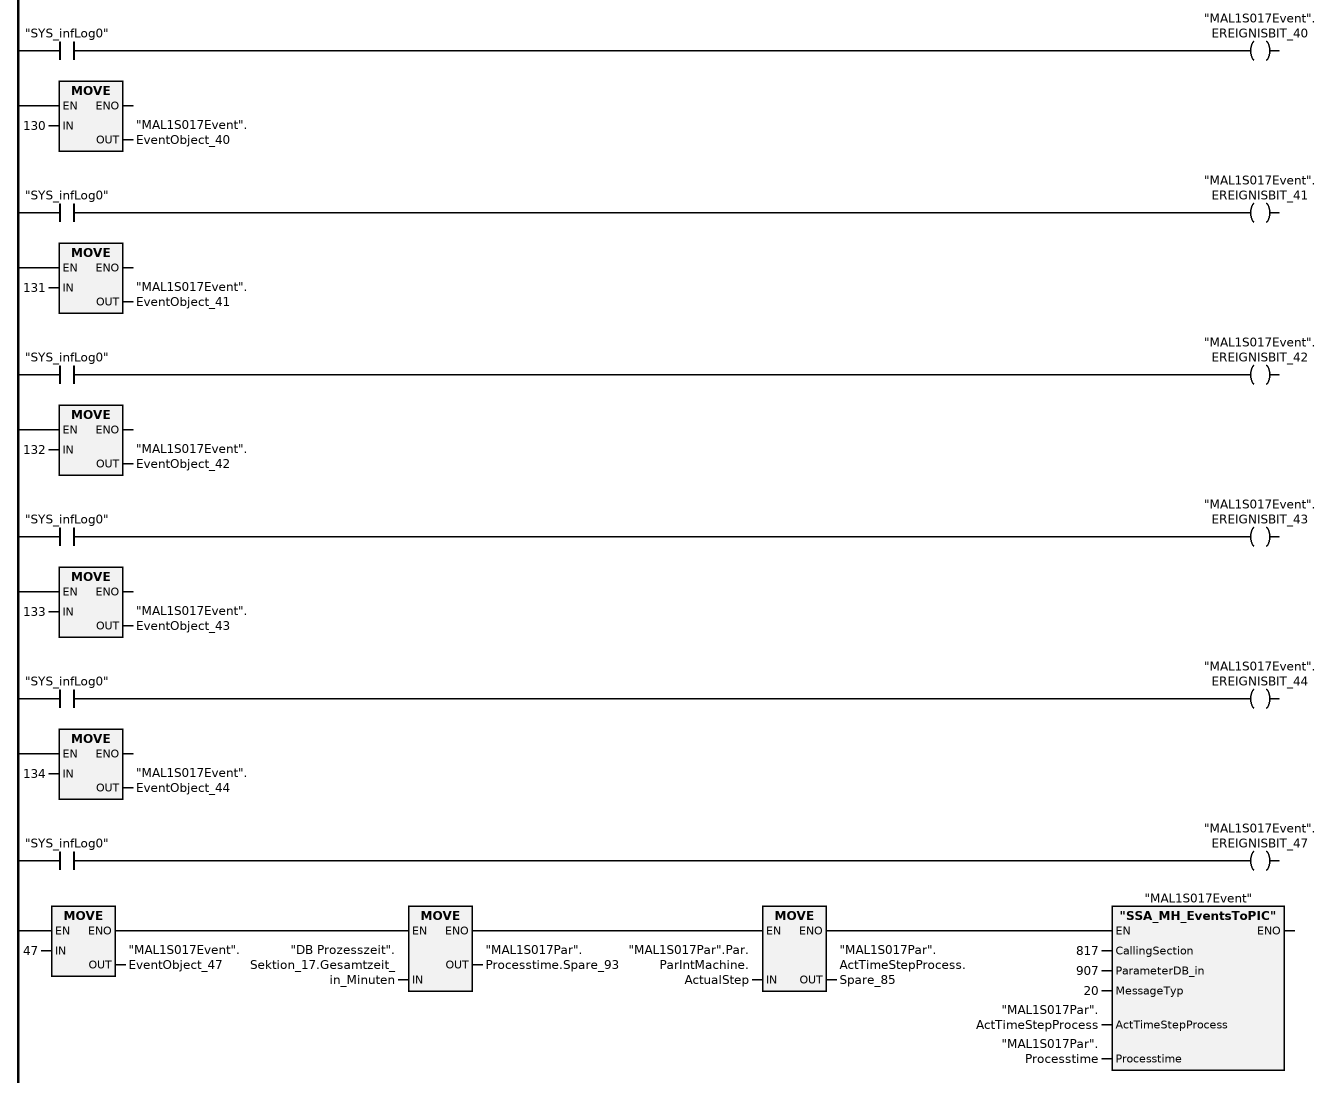
	NOP 0;
	// load events into event input

	// 1. event Process active
	      U     "MAL1S017Par".Par.FlagProcess.ProcessActive;
	      =     "MAL1S017Event".EREIGNISBIT_1;
	      L     1;
	      T     "MAL1S017Event".EventObject_1;
	// 2. event InfDataReady
	      U     "MAL1S017".ToASW.InfDataReady;
	      =     "MAL1S017Event".EREIGNISBIT_2;
	      L     2;
	      T     "MAL1S017Event".EventObject_2;
	// 11. event
	      U     "MAL1S017Par".Par.FlagFunction_1.StepLoading; // Step loading
	      =     "MAL1S017Event".EREIGNISBIT_11;
	      L     1001;
	      T     "MAL1S017Event".EventObject_11;
	// 12. event
	      U     "MAL1S017Par".Par.FlagFunction_1.StepUnloading; // Step Unloading
	      =     "MAL1S017Event".EREIGNISBIT_12;
	      L     1020;
	      T     "MAL1S017Event".EventObject_12;
	// 13. event
	      U     "MAL1S017Par".Par.FlagFunction_1.StepCleaning; // Step Cleaning
	      =     "MAL1S017Event".EREIGNISBIT_13;
	      L     1025;
	      T     "MAL1S017Event".EventObject_13;
	// 14. event
	      U     "MAL1S017Par".Par.FlagProcess2.Turning1WithoutSpraying;
	      O     "MAL1S017Par".Par.FlagProcess2.Turning2WithoutSpraying;
	      =     "MAL1S017Event".EREIGNISBIT_14;
	      L     1046;
	      T     "MAL1S017Event".EventObject_14;
	// 15. event
	      U     "MAL1S017Par".Par.FlagProcess2.Turning1WithSpraying;
	      O     "MAL1S017Par".Par.FlagProcess2.Turning2WithSpraying;
	      =     "MAL1S017Event".EREIGNISBIT_15;
	      L     1049;
	      T     "MAL1S017Event".EventObject_15;
	// 16. event
	      U     "MAL1S017Par".Par.FlagProcess2.Turning1WithDosing;
	      O     "MAL1S017Par".Par.FlagProcess2.Turning2WithDosing;
	      =     "MAL1S017Event".EREIGNISBIT_16;
	      L     1050;
	      T     "MAL1S017Event".EventObject_16;
	// 17. event
	      U     "SYS_infLog0";
	      =     "MAL1S017Event".EREIGNISBIT_17;
	      L     1066;
	      T     "MAL1S017Event".EventObject_17;
	// 18. event
	      U     "SYS_infLog0";
	      =     "MAL1S017Event".EREIGNISBIT_18;
	      L     1048;
	      T     "MAL1S017Event".EventObject_18;
	// 19. event
	      U     "SYS_infLog0";
	      =     "MAL1S017Event".EREIGNISBIT_19;
	      L     109;
	      T     "MAL1S017Event".EventObject_19;
	// 20. event
	      U     "SYS_infLog0";
	      =     "MAL1S017Event".EREIGNISBIT_20;
	      L     110;
	      T     "MAL1S017Event".EventObject_20;
	// 21. event
	      U     "SYS_infLog0";
	      =     "MAL1S017Event".EREIGNISBIT_21;
	      L     111;
	      T     "MAL1S017Event".EventObject_21;
	// 22. event
	      U     "SYS_infLog0";
	      =     "MAL1S017Event".EREIGNISBIT_22;
	      L     112;
	      T     "MAL1S017Event".EventObject_22;
	// 23. event
	      U     "SYS_infLog0";
	      =     "MAL1S017Event".EREIGNISBIT_23;
	      L     113;
	      T     "MAL1S017Event".EventObject_23;
	// 24. event
	      U     "SYS_infLog0";
	      =     "MAL1S017Event".EREIGNISBIT_24;
	      L     114;
	      T     "MAL1S017Event".EventObject_24;
	// 25. event
	      U     "MAL1S017".SecAc.Sta1On.Inf08; // ILO-Mode
	      =     "MAL1S017Event".EREIGNISBIT_25;
	      L     1026;
	      T     "MAL1S017Event".EventObject_25;
	// 26. event
	      U     "SYS_infLog0";
	      =     "MAL1S017Event".EREIGNISBIT_26;
	      L     116;
	      T     "MAL1S017Event".EventObject_26;
	// 27. event
	      U     "SYS_infLog0";
	      =     "MAL1S017Event".EREIGNISBIT_27;
	      L     117;
	      T     "MAL1S017Event".EventObject_27;
	// 28. event
	      U     "SYS_infLog0";
	      =     "MAL1S017Event".EREIGNISBIT_28;
	      L     118;
	      T     "MAL1S017Event".EventObject_28;
	// 29. event
	      U     "SYS_infLog0";
	      =     "MAL1S017Event".EREIGNISBIT_29;
	      L     119;
	      T     "MAL1S017Event".EventObject_29;
	// 30. event
	      U     "SYS_infLog0";
	      =     "MAL1S017Event".EREIGNISBIT_30;
	      L     120;
	      T     "MAL1S017Event".EventObject_30;
	// 31. event
	      U     "SYS_infLog0";
	      =     "MAL1S017Event".EREIGNISBIT_31;
	      L     121;
	      T     "MAL1S017Event".EventObject_31;
	// 32. event
	      U     "SYS_infLog0";
	      =     "MAL1S017Event".EREIGNISBIT_32;
	      L     122;
	      T     "MAL1S017Event".EventObject_32;
	// 33. event
	      U     "SYS_infLog0";
	      =     "MAL1S017Event".EREIGNISBIT_33;
	      L     123;
	      T     "MAL1S017Event".EventObject_33;
	// 34. event
	      U     "SYS_infLog0";
	      =     "MAL1S017Event".EREIGNISBIT_34;
	      L     124;
	      T     "MAL1S017Event".EventObject_34;
	// 35. event
	      U     "SYS_infLog0";
	      =     "MAL1S017Event".EREIGNISBIT_35;
	      L     125;
	      T     "MAL1S017Event".EventObject_35;
	// 36. event
	      U     "SYS_infLog0";
	      =     "MAL1S017Event".EREIGNISBIT_36;
	      L     126;
	      T     "MAL1S017Event".EventObject_36;
	// 37. event
	      U     "SYS_infLog0";
	      =     "MAL1S017Event".EREIGNISBIT_37;
	      L     127;
	      T     "MAL1S017Event".EventObject_37;
	// 38. event
	      U     "SYS_infLog0";
	      =     "MAL1S017Event".EREIGNISBIT_38;
	      L     128;
	      T     "MAL1S017Event".EventObject_38;
	// 39. event
	      U     "SYS_infLog0";
	      =     "MAL1S017Event".EREIGNISBIT_39;
	      L     129;
	      T     "MAL1S017Event".EventObject_39;
	// 40. event
	      U     "SYS_infLog0";
	      =     "MAL1S017Event".EREIGNISBIT_40;
	      L     130;
	      T     "MAL1S017Event".EventObject_40;
	//
	// 41. event
	      U     "SYS_infLog0";
	      =     "MAL1S017Event".EREIGNISBIT_41;
	      L     131;
	      T     "MAL1S017Event".EventObject_41;
	// 42. event
	      U     "SYS_infLog0";
	      =     "MAL1S017Event".EREIGNISBIT_42;
	      L     132;
	      T     "MAL1S017Event".EventObject_42;
	// 43. event
	      U     "SYS_infLog0";
	      =     "MAL1S017Event".EREIGNISBIT_43;
	      L     133;
	      T     "MAL1S017Event".EventObject_43;
	// 44. event
	      U     "SYS_infLog0";
	      =     "MAL1S017Event".EREIGNISBIT_44;
	      L     134;
	      T     "MAL1S017Event".EventObject_44;
	// only for test
	// 47. event
	      U     "SYS_infLog0";
	      =     "MAL1S017Event".EREIGNISBIT_47;
	      L     47;
	      T     "MAL1S017Event".EventObject_47;

	// copy data for event-logging
	      L     "DB Prozesszeit".Sektion_17.Gesamtzeit_in_Minuten;
	      T     "MAL1S017Par".Processtime.Spare_93;
	      L     "MAL1S017Par".Par.ParIntMachine.ActualStep;
	      T     "MAL1S017Par".ActTimeStepProcess.Spare_85;

	//
	      CALL "SSA_MH_EventsToPIC" , "MAL1S017Event" (
	           CallingSection           := 817,
	           ParameterDB_in           := 907,
	           MessageTyp               := 20,
	           ActTimeStepProcess       := "MAL1S017Par".ActTimeStepProcess,
	           Processtime              := "MAL1S017Par".Processtime);
	NETWORK
	TITLE =ASW_6000: Start process germinating
	//
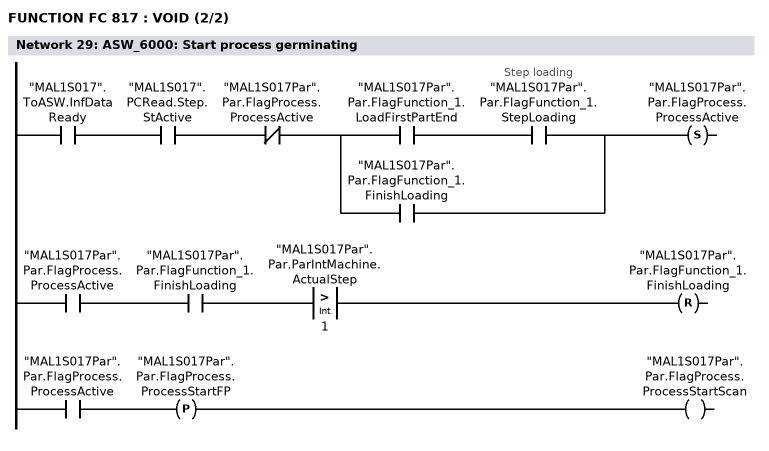
	      U     "MAL1S017".ToASW.InfDataReady;
	      U     "MAL1S017".PCRead.Step.StActive;
	      UN    "MAL1S017Par".Par.FlagProcess.ProcessActive;
	      U(    ;
	//    U     "MAL1S017Par".Par.FlagFunction_1.FinishUnloading
	      U     "MAL1S017Par".Par.FlagFunction_1.LoadFirstPartEnd;
	      U     "MAL1S017Par".Par.FlagFunction_1.StepLoading; // Step loading
	      O     "MAL1S017Par".Par.FlagFunction_1.FinishLoading;
	      )     ;
	      S     "MAL1S017Par".Par.FlagProcess.ProcessActive;

	      U     "MAL1S017Par".Par.FlagProcess.ProcessActive;
	      U     "MAL1S017Par".Par.FlagFunction_1.FinishLoading;
	      U(    ;
	      L     "MAL1S017Par".Par.ParIntMachine.ActualStep;
	      L     1;
	      >I    ;
	      )     ;
	      R     "MAL1S017Par".Par.FlagFunction_1.FinishLoading;
	//
	      U     "MAL1S017Par".Par.FlagProcess.ProcessActive;
	      FP    "MAL1S017Par".Par.FlagProcess.ProcessStartFP;
	      =     "MAL1S017Par".Par.FlagProcess.ProcessStartScan;
	NETWORK
	TITLE =ASW_6010: Process germinating active
	//
	      U     "MAL1S017Par".Par.FlagProcess.ProcessActive;
	      SPBN  E000;
	//-Actual process time---
	      U     "MAL1S017Par".Par.FlagProcess.ProcessStartScan;
	      SPBN  actu;
	      L     1; // Start process first step
	      T     "MAL1S017Par".Par.ParIntMachine.ActualStep;
	      T     "MAL1S017Par".Par.ProcessValue.StepNrActCopy;
	      SPA   newS;
	actu: NOP   0;
	// Prozesszeit
	      L     "DB Prozesszeit".Sektion_17.Tage;
	      INC   1; // malters do not accept day 0!!
	      T     "MAL1S017Par".Processtime.Day;
	      L     "DB Prozesszeit".Sektion_17.Stunden;
	      T     "MAL1S017Par".Processtime.Hour; // Processtime in h
	      L     "DB Prozesszeit".Sektion_17.Minuten;
	      T     "MAL1S017Par".Processtime.Min; // Processtime in min
	      U     "DB Prozesszeit".Sektion_17.Prozess_aktiv; // active bit section 2
	      L      1;
	      SPB    nTa;
	      L      0;
	nTa:  T     "MAL1S017Par".Processtime.ProcessTimeActive;

	// Test new step
	      L     "MAL1S017Par".Par.ParIntMachine.ActualStep;
	      L     "MAL1S017Par".Par.ProcessValue.StepNrActCopy;
	      ==I   ;
	      SPB   oldS;
	newS: NOP   0;
	      L     "MAL1S017Par".Par.ParIntMachine.ActualStep;
	      T     "MAL1S017Par".Par.ProcessValue.StepNrActCopy;
	//
	      L     L#0; // clear actual step time
	      T     "MAL1S017Par".Par.ProcessValue.StepTimeAct; // in ms
	      L     0;
	      T     "MAL1S017Par".ActTimeStepProcess.SteptimeActMinOverall; // Steptime in min overall
	//
	      U(    ;
	      L     "MAL1S017Par".Par.ParIntMachine.ActualStep;
	      L     "MAL1S017".SecNom.GERM.RecipeHeader.NumberOfSteps;
	      >I    ;
	      )     ;
	      SPB   Pend; // last step is finished
	      SET   ;
	      S     "MAL1S017StepValues".StartStep; // start step for average calculating
	      SPA   E000; // to secure, that new step-data are copied
	oldS: NOP   0;
	      L     "ASW_GraphicData".General.CycleTime[1].Actual;
	      L     "MAL1S017Par".Par.ProcessValue.StepTimeAct; // in ms
	      +D    ;
	      T     "MAL1S017Par".Par.ProcessValue.StepTimeAct; // in ms
	      L     "MAL1S017Par".Par.ProcessValue.StepTimeAct; // in ms
	      L     L#86400000; // ms/d
	      MOD   ;
	      L     L#3600000; // ms/h
	      /D    ;
	      T     "MAL1S017Par".ActTimeStepProcess.SteptimeActHour; // Steptime in h
	//
	      L     "MAL1S017Par".Par.ProcessValue.StepTimeAct;
	      L     L#3600000; // ms/h
	      MOD   ;
	      L     L#60000; // ms/min
	      /D    ;
	      T     "MAL1S017Par".ActTimeStepProcess.SteptimeActMin; // Steptime in min
	//
	      L     "MAL1S017Par".Par.ProcessValue.StepTimeAct;
	      L     L#60000; // ms/min
	      /D    ;
	      T     "MAL1S017Par".ActTimeStepProcess.SteptimeActMinOverall; // Steptime in min overall
	//
	// Next Step
	//
	//  Switch over to next step under conditions:
	//  or Maximal steptime
	//  or Minimal steptime
	//          and
	//              or no setpoint delta temp
	//              or atual value delta temp is ge setpoint deltatemp
	//                  and sensor is ok
	//          and
	//              or no setpoint max temp above floor
	//              or atual value max temp above floor is ge setpoint max temp above floor
	//                  and sensor is ok

	// Total hours 0..32767
	      L     "MAL1S017Par".ActTimeStepProcess.SteptimeActMinOverall; // Steptime in min overall
	      ITD   ;
	      DTR   ;
	      L     6.000000e+001; // min/h
	      /R    ;
	      TRUNC ;
	      T     "MAL1S017Par".ActTimeStepProcess.StepTimeActHourTotal; // Steptime in hours overall
	//
	// 1 Kriterium - steptime minimal
	      U(    ;
	      L     "MAL1S017Par".ActTimeStepProcess.StepTimeActHourTotal; // Steptime in hours overall
	      L     "MAL1S017Par".StepAct.StepTime_Min; // Target steptime actual step
	      >=I   ;
	      )     ;
	      U(    ; // and  one of
	// 2 Kriterium - or delta temperature
	      O(    ;
	      UN     G103M.A_2191_BTE02.OutOverflow; //AIR TEMPERATURE ABOVE FLOOR
	      UN     G103M.A_2191_BTE02.OutFaultAI; //AIR TEMPERATURE ABOVE FLOOR
	      UN     G103M.A_2191_BTE01.OutOverflow; //AIR TEMPERATURE BELOW FLOOR
	      UN     G103M.A_2191_BTE01.OutFaultAI; //AIR TEMPERATURE BELOW FLOOR
	      U     "MAL1S017Par".Par.FlagProcess1.DeltaTempNextStep;
	      U(    ;
	      L     "MAL1S017Par".Par.ProcessValue.ActValueDeltaTempDint;
	      L     "MAL1S017Par".StepAct.DeltaTempSwitchpointStep;
	      >=D   ;
	      )     ;
	      )     ;
	// 3 Kriterium - or setpoint temperature above floor
	      O(    ;
	      UN     G103M.A_2191_BTE02.OutOverflow; //AIR TEMPERATURE ABOVE FLOOR
	      UN     G103M.A_2191_BTE02.OutFaultAI; //AIR TEMPERATURE ABOVE FLOOR
	      U     "MAL1S017Par".Par.FlagProcess1.MaxTempNextStep;
	      U(    ;
	      L     "MAL1S017Par".Par.ProcessValue.ActValMaxTempAboveDint;
	      L     "MAL1S017Par".StepAct.MaxTempAboveFloorStep;
	      >=D   ;
	      )     ;
	      )     ;
	      )     ;
	// 4 Kriterium - or only maimal steptime
	      O(    ;
	      L     "MAL1S017Par".ActTimeStepProcess.StepTimeActHourTotal; // Steptime in hours overall
	      L     "MAL1S017Par".StepAct.StepTime_Max; // Target steptime actual step
	      >=I   ;
	      )     ;
	      SPBN  E000;

	// send average step data to PIC
	      SET   ;
	      S     "MAL1S017StepValues".SendData; // send average step data to PIC
	// Next step
	      L     "MAL1S017Par".Par.ParIntMachine.ActualStep;
	      L     "MAL1S017".SecNom.GERM.RecipeHeader.NumberOfSteps;
	      >I    ;
	      SPB   Pend; // Last step is finished
	//
	      L     "MAL1S017Par".Par.ParIntMachine.ActualStep;
	      L     1;
	      +I    ;
	      T     "MAL1S017Par".Par.ParIntMachine.ActualStep;
	      L     0;
	      T     "MAL1S017Par".ActTimeStepProcess.SteptimeActMinOverall; // Steptime in min overall
	      SET   ;
	      R     "MAL1S017Par".Par.FlagProcess.MessageNoNextStep; // Meldung "No next step"
	      SPA   E000;
	Pend: NOP   0; // Process has finished
	      SET   ;
	      R     "MAL1S017Par".Par.FlagProcess.ProcessActive;
	      S     "MAL1S017Par".Par.FlagProcess.ProcessEnd; // germinating Process finished
	//
	      L     0; // clear step number
	      T     "MAL1S017Par".Par.ParIntMachine.ActualStep;
	E000: NOP   0;

	NETWORK
	TITLE =ASW_6030: Active step germinating
	//      U     "MAL1S017Par".Par.FlagProcess.ProcessActive;
	//      SPBN  tuen;
	//
	//	// copy stepnr
	//	      L     "MAL1S017Par".Par.ParIntMachine.ActualStep;
	//	      T     "MAL1S017Par".Par.ParIntProcess.ActualStep;
	//	// set step conditions
	//
	//	// Case where process is starting during loading
	//	      U     "MAL1S017Par".Par.FlagProcess.ProcessActive;
	//	      UN    "MAL1S017Par".Par.FlagFunction_1.StepLoading; // Step loading
	//	      SPBN  e003;
	//	// lifting devices must be in highest position
	//	      L       WinCoS_BIW01_09PLC1BIW01_02.Ma.Par.ParPositionTopRightUnits; //Malting Plant OAO Belsolod Ivanonvo Weissrussland
	//	      L     50; // 50mm offset
	//	      +I    ;
	//	      T     "MAL1S017Par".Par.MachineValue.SOLLWERT_HUBZUG1_HOEHE;
	//	      L       WinCoS_BIW01_09PLC1BIW01_02.Ma.Par.ParPositionTopLeftUnits; //Malting Plant OAO Belsolod Ivanonvo Weissrussland
	//	      L     50; // 50mm offset
	//	      +I    ;
	//	      T     "MAL1S017Par".Par.MachineValue.SOLLWERT_HUBZUG2_HOEHE;
	//	      L     5;
	//	      T     WinCoS_BIW01_09PLC1BIW01_02.Ma.Par.ParTolPosition;
	//	e003: NOP   0;
	//
	//	// reset turning cmds
	//
	//	// save turning cmds from prev.step
	//	      L     "MAL1S017Par".Par.ParIntMachine.ActualStep;
	//	      L     "MAL1S017Par".Par.ParIntProcess.PrevStep1stTurn;
	//	      <>I   ;
	//	      SPB   sav1;
	//	      U     "MAL1S017Par".Par.FlagProcess2.Turning1WithSpraying;
	//	      =     "MAL1S017Par".Par.Switches1.StaOn08; // Turning1WithSpraying
	//	      U     "MAL1S017Par".Par.FlagProcess2.Turning1WithDosing;
	//	      =     "MAL1S017Par".Par.Switches1.StaOn09; // Turning1WithDosing
	//	sav1: NOP   0;
	//	      L     "MAL1S017Par".Par.ParIntMachine.ActualStep;
	//	      L     "MAL1S017Par".Par.ParIntProcess.PrevStep2ndTurn;
	//	      <>I   ;
	//	      SPB   sav2;
	//	      U     "MAL1S017Par".Par.FlagProcess2.Turning2WithSpraying;
	//	      =     "MAL1S017Par".Par.Switches1.StaOn10; // Turning2WithSpraying
	//	      U     "MAL1S017Par".Par.FlagProcess2.Turning2WithDosing;
	//	      =     "MAL1S017Par".Par.Switches1.StaOn11; // Turning2WithDosing
	//	sav2: NOP   0;
	//
	//	      SET   ;
	//	      R     "MAL1S017Par".Par.FlagProcess2.Turning1WithoutSpraying;
	//	      R     "MAL1S017Par".Par.FlagProcess2.Turning1WithSpraying;
	//	      R     "MAL1S017Par".Par.FlagProcess2.Turning1WithDosing;
	//	      R     "MAL1S017Par".Par.FlagProcess2.Turning2WithoutSpraying;
	//	      R     "MAL1S017Par".Par.FlagProcess2.Turning2WithSpraying;
	//	      R     "MAL1S017Par".Par.FlagProcess2.Turning2WithDosing;
	//
	//	// Delta Temp to switch to next step
	//	      L     "MAL1S017Par".StepAct.DeltaTempSwitchpointStep;
	//	      L     L#0;
	//	      >D   ;
	//	      =     "MAL1S017Par".Par.FlagProcess1.DeltaTempNextStep;
	//	// Max Temp to switch to next step
	//	      L     "MAL1S017Par".StepAct.MaxTempAboveFloorStep;
	//	      L     L#0;
	//	      >D   ;
	//	      =     "MAL1S017Par".Par.FlagProcess1.MaxTempNextStep;
	//
	//	// position waste air see sub 6050
	//
	//	// basic speed fan see sub 6040
	//
	//	// air humifidication
	//	      L     1;
	//	      L     "MAL1S017Par".StepAct.AirMoisten;   // On/Off
	//	      ==I;  // air humifidication on
	//	      U     G105M.A_2160_MXZ01.Ma.StStartedFwd; //TRAVELING DRIVE
	//	      =     "MAL1S017Par".Par.FlagProcess.AirHumidificationValve1; // air humifidication valve 1 on
	//	      U(    ; // air humifidication on
	//	      L     "MAL1S017Par".Par.ParIntMachine.TargetSpeedGermFan; // germinating fan is running
	//	      L     40; // fanspeed > 40%
	//	      >I    ; // muss noch in Istwert getauscht werden JV
	//	      )     ; // fanspeed > 40%
	//	      =     "MAL1S017Par".Par.FlagProcess.AirHumidificationValve2;
	//
	//	// air cooling
	//	      L     "MAL1S017Par".StepAct.Cooling;
	//	      L   1;  // Activate Cooling System = 1 (yes)
	//	      ==I;
	//	      =     "MAL1S017Par".Par.FlagProcess.Cooling; // request cooling
	//
	//	      U     "MAL1S017Par".Par.FlagProcess.ProcessActive;
	//	      U     "MAL1S017".PCRead.Step.StReady;
	//	      UN    "MAL1S017Par".Par.FlagFunction_1.StepLoading;
	//	      SPBN  e630;
	//
	//	// turning 1
	//	      UN    "MAL1S017Par".Par.FlagProcess2.StartSecondTurningRound; // Turn from PrevStep
	//	      U(;
	//	      L     "MAL1S017Par".StepAct.StartTurningRound_1;
	//	      L     0;
	//	      >=D;                  // negative, no turning 1
	//	      );
	//	      U(    ;
	//	      O(    ; // Nach Rezept
	//	      L     "MAL1S017Par".ActTimeStepProcess.StepTimeActHourTotal; // Steptime in hours overall
	//	      L     "MAL1S017Par".StepAct.StartTurningRound_1;
	//	      ==I   ;
	//      UN     G100M.A_2111_MXZ41MA.Ma.StAdjusted; // target position turning reached
	//      )     ;
	//      O(    ; // Selbsthaltung
	//      L     "MAL1S017Par".ActTimeStepProcess.StepTimeActHourTotal; // Steptime in hours overall
	//      L     "MAL1S017Par".StepAct.StartTurningRound_1;
	//      <>I   ;
	//      U     "MAL1S017Par".Par.FlagProcess2.StartFirstTurningRound;
	//      )     ;
	//      )     ;
	//      S     "MAL1S017Par".Par.FlagProcess2.Turning1WithoutSpraying;
	//      S     "MAL1S017Par".Par.FlagFunction_1.TurningStart;
	//// turning 1 with spraying
	//      U(    ;
	//      L     1;
	//      L     "MAL1S017Par".StepAct.TurningWithSpraying_1;
	//      ==I;    // turning 1 with spraying on
	//      U(    ;
	//      L     "MAL1S017Par".Par.ParIntMachine.ActualStep;
	//      L     "MAL1S017Par".Par.ParIntProcess.PrevStep1stTurn;
	//      ==I   ;
	//      )     ;
	//      )     ;
	//      O(    ;
	//      L     "MAL1S017Par".Par.ParIntMachine.ActualStep;
	//      L     "MAL1S017Par".Par.ParIntProcess.PrevStep1stTurn;
	//      <>I   ;
	//      U     "MAL1S017Par".Par.Switches1.StaOn08; // Turning1WithSpraying
	//      )     ;
	//      U     "MAL1S017Par".Par.FlagProcess2.Turning1WithoutSpraying;
	//      S     "MAL1S017Par".Par.FlagProcess2.Turning1WithSpraying;
	//// turning 1 with spraying and GA3
	//      U(    ;
	//      L     1;
	//      L     "MAL1S017Par".StepAct.TurningWithDosing_1;
	//      ==I;    // turning 1 with spraying on
	//      U(    ;
	//      L     "MAL1S017Par".Par.ParIntMachine.ActualStep;
	//      L     "MAL1S017Par".Par.ParIntProcess.PrevStep1stTurn;
	//      ==I   ;
	//      )     ;
	//      )     ;
	//      O(    ;
	//      L     "MAL1S017Par".Par.ParIntMachine.ActualStep;
	//      L     "MAL1S017Par".Par.ParIntProcess.PrevStep1stTurn;
	//      <>I   ;
	//      U     "MAL1S017Par".Par.Switches1.StaOn09; // Turning1WithDosing
	//      )     ;
	//      U     "MAL1S017Par".Par.FlagProcess2.Turning1WithoutSpraying;
	//      S     "MAL1S017Par".Par.FlagProcess2.Turning1WithSpraying;
	//      S     "MAL1S017Par".Par.FlagProcess2.Turning1WithDosing;
	//
	//      U     "MAL1S017Par".Par.FlagProcess2.Turning1WithoutSpraying;
	//      U     "MAL1S017Par".Par.FlagFunction_1.TurningStart;
	//      UN     G100M.A_2111_MXZ41MA.Ma.StAdjusted; // target position turning reached
	//      FP    "MAL1S017Par".Par.FlagProcess2.StartFirstTurningFP;
	//      S     "MAL1S017Par".Par.FlagProcess2.StartFirstTurningRound;
	//
	//      U     G100M.A_2111_MXZ41MA.Ma.StAdjusted; // target position turning reached
	//      O(    ;
	//      L     "MAL1S017Par".ActTimeStepProcess.StepTimeActHourTotal; // Steptime in hours overall
	//      L     "MAL1S017Par".StepAct.StartTurningRound_1;
	//      >I    ;
	//      U     G100M.A_2111_MXZ41MA.Ma.StAdjusted; // target position turning reached
	//      )     ;
	//      U     "MAL1S017Par".Par.FlagProcess2.StartFirstTurningRound;
	//      R     "MAL1S017Par".Par.FlagProcess2.StartFirstTurningRound;
	//
	//      U     "MAL1S017Par".Par.FlagProcess2.StartFirstTurningFP;
	//      SPB   trn1;
	//      L     "MAL1S017Par".Par.ParIntMachine.ActualStep;
	//      T     "MAL1S017Par".Par.ParIntProcess.PrevStep1stTurn;
	//trn1: NOP   0;
	//
	//// turning 2
	//      UN    "MAL1S017Par".Par.FlagProcess2.StartFirstTurningRound; // Unsinngie Rezeptwerte
	//      U(;
	//      L     1;
	//      L     "MAL1S017Par".StepAct.StartTurningRound_2;
	//      ==I    ;
	//      );
	//      U(    ;
	//      O(    ; // Nach Rezept
	//      L     "MAL1S017Par".ActTimeStepProcess.StepTimeActHourTotal; // Steptime in hours overall
	//      L     "MAL1S017Par".StepAct.StartTurningRound_2;
	//      ==I   ;
	//      UN     G100M.A_2111_MXZ41MA.Ma.StAdjusted; // target position turning reached
	//      )     ;
	//      O(    ; // Selbsthaltung
	//      L     "MAL1S017Par".ActTimeStepProcess.StepTimeActHourTotal; // Steptime in hours overall
	//      L     "MAL1S017Par".StepAct.StartTurningRound_2;
	//      <>I   ;
	//      U     "MAL1S017Par".Par.FlagProcess2.StartSecondTurningRound;
	//      )     ;
	//      )     ;
	//      S     "MAL1S017Par".Par.FlagProcess2.Turning2WithoutSpraying;
	//      S     "MAL1S017Par".Par.FlagFunction_1.TurningStart;
	//// turning 2 with spraying
	//      U(    ;
	//      L     1;
	//      L     "MAL1S017Par".StepAct.TurningWithSpraying_2;
	//      ==I    ;
	//      U(    ;
	//      L     "MAL1S017Par".Par.ParIntMachine.ActualStep;
	//      L     "MAL1S017Par".Par.ParIntProcess.PrevStep2ndTurn;
	//      ==I   ;
	//      )     ;
	//      )     ;
	//      O(    ;
	//      L     "MAL1S017Par".Par.ParIntMachine.ActualStep;
	//      L     "MAL1S017Par".Par.ParIntProcess.PrevStep2ndTurn;
	//      <>I   ;
	//      U     "MAL1S017Par".Par.Switches1.StaOn10; // Turning2WithSpraying
	//      )     ;
	//      U     "MAL1S017Par".Par.FlagProcess2.Turning2WithoutSpraying;
	//      S     "MAL1S017Par".Par.FlagProcess2.Turning2WithSpraying;
	//// turning 2 with spraying and GA3
	//      U(    ;
	//      L     1;
	//      L     "MAL1S017Par".StepAct.TurningWithDosing_2;
	//      ==I;    // turning 2 with spraying and GA3 on
	//      U(    ;
	//      L     "MAL1S017Par".Par.ParIntMachine.ActualStep;
	//      L     "MAL1S017Par".Par.ParIntProcess.PrevStep2ndTurn;
	//      ==I   ;
	//      )     ;
	//      )     ;
	//      O(    ;
	//      L     "MAL1S017Par".Par.ParIntMachine.ActualStep;
	//      L     "MAL1S017Par".Par.ParIntProcess.PrevStep2ndTurn;
	//      <>I   ;
	//      U     "MAL1S017Par".Par.Switches1.StaOn11; // Turning2WithDosing
	//      )     ;
	//      U     "MAL1S017Par".Par.FlagProcess2.Turning2WithoutSpraying;
	//      S     "MAL1S017Par".Par.FlagProcess2.Turning2WithSpraying;
	//      S     "MAL1S017Par".Par.FlagProcess2.Turning2WithDosing;
	//
	//      U     "MAL1S017Par".Par.FlagProcess2.Turning2WithoutSpraying;
	//      U     "MAL1S017Par".Par.FlagFunction_1.TurningStart;
	//      UN     G100M.A_2111_MXZ41MA.Ma.StAdjusted; // target position turning reached
	//      FP    "MAL1S017Par".Par.FlagProcess2.StartSecondTurningFP;
	//      S     "MAL1S017Par".Par.FlagProcess2.StartSecondTurningRound;
	//
	//      U     G100M.A_2111_MXZ41MA.Ma.StAdjusted; // target position turning reached
	//      O(    ;
	//      L     "MAL1S017Par".ActTimeStepProcess.StepTimeActHourTotal; // Steptime in hours overall
	//      L     "MAL1S017Par".StepAct.StartTurningRound_2;
	//      >I    ;
	//      U     G100M.A_2111_MXZ41MA.Ma.StAdjusted; // target position turning reached
	//      )     ;
	//      U     "MAL1S017Par".Par.FlagProcess2.StartSecondTurningRound;
	//      R     "MAL1S017Par".Par.FlagProcess2.StartSecondTurningRound;
	//
	//      U     "MAL1S017Par".Par.FlagProcess2.StartSecondTurningFP;
	//      SPB   trn2;
	//      L     "MAL1S017Par".Par.ParIntMachine.ActualStep;
	//      T     "MAL1S017Par".Par.ParIntProcess.PrevStep2ndTurn;
	//trn2: NOP   0;
	////Fix Speed for Turning
	//      U     "MAL1S017Par".Par.FlagProcess2.Turning1WithoutSpraying;
	//      O     "MAL1S017Par".Par.FlagProcess2.Turning1WithSpraying;
	//      O     "MAL1S017Par".Par.FlagProcess2.Turning2WithoutSpraying;
	//      O     "MAL1S017Par".Par.FlagProcess2.Turning2WithSpraying;
	//      U    M 50.0;
	//      SPBN  SpdT;
	//      L     15; // 15Hz
	//      T     "MAL1S017Par".Par.MachineValue.SollwertFahrantrieb;
	//SpdT: NOP   0;
	//
	//// find turning direction
	//      U     "MAL1S017Par".Par.FlagGen.TurningStarted;
	//      O(    ;
	//      UN    "MAL1S017Par".Par.FlagProcess2.Turning1WithoutSpraying;
	//      UN    "MAL1S017Par".Par.FlagProcess2.Turning2WithoutSpraying;
	//      )     ;
	//      SPB   tuen;
	//      L     "MAL1S017Par".Par.ParIntMachine.TargetPosTravDriTurnRigt; // 370° = endposition turning right
	//      T     G100M.A_2111_MXZ41MA.Ma.InPositionTarget; // target position turning reached
	//
	//      U(    ;
	//      L     G100M.A_2111_MXZ41MA.Ma.OutPositionAngle;
	//      L     1800;
	//      <I    ; // condition turning right (clockwise)
	//      )     ;
	//      S     "MAL1S017Par".Par.FlagFunction_1.TurningRight;
	//      S     "MAL1S017Par".Par.FlagGen.TurningStarted;
	//// - Correct effect of ILO Mode
	//      L       WinCoS_BIW01_09PLC1BIW01_02.Ma.Par.ParPositionTopLeftUnits; //Malting Plant OAO Belsolod Ivanonvo Weissrussland
	//      T     "MAL1S017Par".Par.MachineValue.SOLLWERT_HUBZUG1_HOEHE;
	//      L       WinCoS_BIW01_09PLC1BIW01_02.Ma.Par.ParPositionTopRightUnits; //Malting Plant OAO Belsolod Ivanonvo Weissrussland
	//      T     "MAL1S017Par".Par.MachineValue.SOLLWERT_HUBZUG2_HOEHE;
	//      SPB   E603   ;
	//      L     "MAL1S017Par".Par.ParIntMachine.TargetPosTravDriTurnLeft; // 0° = endposition turning left
	//      T     G100M.A_2111_MXZ41MA.Ma.InPositionTarget; // target position turning reached
	//
	//      U(    ;
	//      L     G100M.A_2111_MXZ41MA.Ma.OutPositionAngle;
	//      L     1800;
	//      >=I   ; // condition turning left (counterclockwise)
	//      )     ;
	//      S     "MAL1S017Par".Par.FlagFunction_1.TurningLeft;
	//      S     "MAL1S017Par".Par.FlagGen.TurningStarted;
	//// - Correct effect of ILO Mode
	//      L       WinCoS_BIW01_09PLC1BIW01_02.Ma.Par.ParPositionTopLeftUnits; //Malting Plant OAO Belsolod Ivanonvo Weissrussland
	//      T     "MAL1S017Par".Par.MachineValue.SOLLWERT_HUBZUG1_HOEHE;
	//      L       WinCoS_BIW01_09PLC1BIW01_02.Ma.Par.ParPositionTopRightUnits; //Malting Plant OAO Belsolod Ivanonvo Weissrussland
	//      T     "MAL1S017Par".Par.MachineValue.SOLLWERT_HUBZUG2_HOEHE;
	//      SPB   E603   ;
	//tuen: NOP   0;
	//// - Case of fast speed to protect a 2nd start during same hours as finsihed
	//      O(    ; // Nach Rezept
	//      L     "MAL1S017Par".ActTimeStepProcess.StepTimeActHourTotal; // Steptime in hours overall
	//      L     "MAL1S017Par".StepAct.StartTurningRound_1;
	//      ==I   ;
	//      U     G100M.A_2111_MXZ41MA.Ma.StAdjusted; // target position turning reached
	//      U     "MAL1S017Par".Par.FlagFunction_1.TurningStart;
	//      )     ;
	//      O(    ; // Nach Rezept
	//      L     "MAL1S017Par".ActTimeStepProcess.StepTimeActHourTotal; // Steptime in hours overall
	//      L     "MAL1S017Par".StepAct.StartTurningRound_2;
	//      ==I   ;
	//      U     G100M.A_2111_MXZ41MA.Ma.StAdjusted; // target position turning reached
	//      U     "MAL1S017Par".Par.FlagFunction_1.TurningStart;
	//      )     ;
	//      SPB   e603;
	//
	//// reset turning right (clockwise)
	//      U     "MAL1S017Par".Par.FlagFunction_1.TurningRight;
	//      U(    ;
	//      O      G100M.A_2111_MXZ41MA.Ma.StAdjusted; // target position turning reached
	//      O(    ;
	//      L     G100M.A_2111_MXZ41MA.Ma.OutPositionAngle;
	//      L     G100M.A_2111_MXZ41MA.Ma.Par.ParTolPosition;
	//      +I    ;
	//      L     "MAL1S017Par".Par.ParIntMachine.TargetPosTravDriTurnRigt;
	//      >=I   ;
	//      )     ;
	//      )     ;
	//      R     "MAL1S017Par".Par.FlagFunction_1.TurningRight;
	//      R     "MAL1S017Par".Par.FlagFunction_1.TurningStart;
	//
	//// reset turning left (counterclockwise)
	//      U     "MAL1S017Par".Par.FlagFunction_1.TurningLeft;
	//      U(    ;
	//      O     G100M.A_2111_MXZ41MA.Ma.StAdjusted; // target position turning reached
	//      O(    ;
	//      L     G100M.A_2111_MXZ41MA.Ma.OutPositionAngle;
	//      L     G100M.A_2111_MXZ41MA.Ma.Par.ParTolPosition;
	//      -I    ;
	//      L     "MAL1S017Par".Par.ParIntMachine.TargetPosTravDriTurnLeft;
	//      <=I   ;
	//      )     ;
	//      )     ;
	//      R     "MAL1S017Par".Par.FlagFunction_1.TurningLeft;
	//      R     "MAL1S017Par".Par.FlagFunction_1.TurningStart;
	//
	//// reset turning flag
	//      U     "MAL1S017Par".Par.FlagGen.TurningStarted;
	//      UN    "MAL1S017Par".Par.FlagProcess2.Turning1WithoutSpraying;
	//      UN    "MAL1S017Par".Par.FlagProcess2.Turning2WithoutSpraying;
	//      O(    ;
	//      U     "MAL1S017Par".Par.FlagGen.TurningStarted;
	//      U     G100M.A_2111_MXZ41MA.Ma.StAdjusted; // target position turning reached
	//      )     ;
	//      ON    "MAL1S017Par".Par.FlagProcess.ProcessActive;
	//      R     "MAL1S017Par".Par.FlagGen.TurningStarted;
	//      R     "MAL1S017Par".Par.FlagProcess2.Turning1WithoutSpraying;
	//      R     "MAL1S017Par".Par.FlagProcess2.Turning2WithoutSpraying;
	//      R     "MAL1S017Par".Par.FlagFunction_1.TurningStart;
	//e630: NOP   0;
	//      UN    "MAL1S017Par".Par.FlagProcess.ProcessActive;
	//      R     "MAL1S017Par".Par.FlagProcess2.StartFirstTurningRound;
	//      R     "MAL1S017Par".Par.FlagProcess2.StartSecondTurningRound;
	//
	//e603: NOP   0;
	//E603: NOP   0;
	NETWORK
	TITLE =ASW_6040: Set fanspeed by delta-t
	//Die Drehzahl des Ventilators wird zwischen dem Rezeptsollwert, als Untere
	//Grenze, und 100% oder Rezeptsollwert, als obere Grenze, geregelt. Die Regelung
	//erfolgt nach folgendem Prinzip:
	//"Delta-T" ist die Differenz zwischen der Soll-Temperatur (Rezeptsollwert) unter
	//der Horde und der gemessenen Ist-Temperatur über der Horde.
	//Steigt die Ist-Temperatur über der Horde und "Delta-T" wird > als der Sollwert
	//im Rezept, so wird die Drehzahl des Ventilators stufenweise erhöht. Maximale
	//Drehzahl ist 100% oder Rezeptsollwert.
	//Sinkt die Ist-Temperatur über der Horde und "Delta-T" wird < als der Sollwert
	//im
	//Rezept, so wird die Drehzahl des Ventilators stufenweise verringert. Minimale
	//Drehzahl ist der Rezeptsollwert.
	//Die Rampen (Stufen) werden durch den Technologen festgelegt und in Programmcode
	//eingetragen. Es sind keine Rezeptsollwerte.
	      NOP   0;
	// recipe setpoint
	      L     "MAL1S017Par".Par.ProcessValue.StepTimeAct; // in ms
	      L     L#1000; // in first secunde steptime
	      >D    ;
	      SPB   regu;
	      SPA   Summ;
	regu: NOP   0;

	      U     "MAL1S017".ToASW.CmdModify;
	      SPB   Summ;

	// Setpoint
	      L     "MAL1S017Par".StepAct.TemperaturAboveFloor;
	      L     "MAL1S017Par".StepAct.TemperaturBelowFloor;
	      -D    ;
	      T     "MAL1S017Par".Par.ProcessValue.SetpointDeltaTempDint;
	// actual value
	      L     G103M.A_2191_BTE02.OutValueUnits; //AIR TEMPERATURE ABOVE FLOOR
	      L     L#10; // von xx,xx°C AUF xx,x°C
	      /D    ;
	      L     "MAL1S017Par".StepAct.TemperaturBelowFloor;
	      -D    ;
	      T     "MAL1S017Par".Par.ProcessValue.ActValueDeltaTempDint;
	// flags to inc/dec
	      L     "MAL1S017Par".Par.ProcessValue.SetpointDeltaTempDint;
	      -D    ;
	      T     "MAL1S017Par".Par.ProcessValue.ResultDeltaTemp;
	      L     L#0;
	      >D    ;
	      =     "MAL1S017Par".Par.FlagProcess1.DeltaTempPlus;
	      <D    ;
	      =     "MAL1S017Par".Par.FlagProcess1.DeltaTempMinus;

	      U     "MAL1S017Par".Par.FlagProcess1.DeltaTempPlus;
	      U     "SYS_Scan0_Tick1min";
	      SPBN  dec;
	      L     "MAL1S017Par".Par.ParIntMachine.TargetSpeedGermFan;
	      L     100; // linmit max
	      >=I   ;
	      SPB   dec;
	      L     "MAL1S017Par".Par.ParIntMachine.TargetSpeedGermFan;
	      L     1;
	      +I    ;
	      T     "MAL1S017Par".Par.ParIntMachine.TargetSpeedGermFan;
	      SPA   e604;
	dec:  NOP   0;
	      U     "MAL1S017Par".Par.FlagProcess1.DeltaTempMinus;
	      U     "SYS_Scan0_Tick1min";
	      SPBN  e604;
	      L     "MAL1S017Par".Par.ParIntMachine.TargetSpeedGermFan;
	      L     "MAL1S017Par".StepAct.SpeedVentilatorBasic; // linmit min
	      <=I   ;
	      SPB   e604;
	      L     "MAL1S017Par".Par.ParIntMachine.TargetSpeedGermFan;
	      L     1;
	      -I    ;
	      T     "MAL1S017Par".Par.ParIntMachine.TargetSpeedGermFan;
	      SPA   e604;

	Summ: NOP   0;
	      L     "MAL1S017Par".StepAct.SpeedVentilatorBasic;
	      T     "MAL1S017Par".Par.ParIntMachine.TargetSpeedGermFan;
	e604: NOP   0;
	E604: NOP   0;
	NETWORK
	TITLE =ASW_6050: Position waste air
	//Der Betriebsart Sommerbetrieb/Winterbetrieb wird durch den Bediener per Rezept
	//bestimmt.
	//Wird die Kühlung im Rezept angewählt, so erfolgt die Umschaltung AUF
	//Sommerbetrieb. Die Frischluftklappe wird nach dem Rezeptsollwert gestellt.
	//Es erfolgt keine Regelung.
	//Wird die Kühlung im Rezept abgewählt, so erfolgt die Umschaltung AUF
	//Winterbetrieb. Die Frischluftklappe wird zuerst nach dem Rezeptsollwert
	//gestellt. Der Rezeptsollwert ist die untere Grenze für die Regelung.
	//Wird die Soll-Temperatur unter der Horde von Kühl- Heizanlage nicht eingehalten
	//-Temperatur zu hoch und der Schaltpunkt überschritten, so wird die
	//Frischluftklappe stufenweise geöffnet.
	//Maximalwert ist 100%.
	//Wird die Soll-Temperatur unter der Horde von Kühl- Heizanlage nicht eingehalten
	//-Temperatur zu niedrig und der Schaltpunkt unterschritten, so wird die
	//Frischluftklappe stufenweise geschlossen.
	//Minimalwert ist der Rezeptsollwert.
	       NOP 0;
	// setpoint waste air
	      U M 50.0;
	      = M 50.0;
	      L     L#10; // 1,0°
	      T     "MAL1S017Par".StepAct.DeltaTempSwitchpointAir;

	// recipe setpoint
	      L     "MAL1S017Par".Par.ProcessValue.StepTimeAct; // in ms
	      L     L#1000; // in first secunde steptime
	      >D    ;
	      SPB   Reg;
	      SPA   summ;
	Reg:  NOP   0;

	// Cooling or heating from cooling defive active --> no flap regulation!
	      U M 50.0;
	//      U     "ComDB_Cooling".Ma.ACK.ActivFlag.Cool.Germinating_1_Started // Internal or external coooling is running
	      O     "MAL1S017".ToASW.CmdModify;
	      SPB   summ;

	      L        G103M.A_2191_BTE01.OutValueUnits; //AIR TEMPERATURE BELOW FLOOR
	      L     L#10; // von xx,xx°C AUF xx,x°C
	      /D    ;
	      L     "MAL1S017Par".StepAct.TemperaturBelowFloor;
	      -D    ;
	      L     "MAL1S017Par".StepAct.DeltaTempSwitchpointAir;
	      >D    ;
	      =     "MAL1S017Par".Par.FlagProcess1.FreshAirFlapOPEN;

	      L        G103M.A_2191_BTE01.OutValueUnits; //AIR TEMPERATURE BELOW FLOOR
	      L     L#10; // von xxx,xx°C AUF xxx,x°C
	      /D    ;
	      L     "MAL1S017Par".StepAct.TemperaturBelowFloor;
	      TAK   ;
	      -D    ;
	      L     "MAL1S017Par".StepAct.DeltaTempSwitchpointAir;
	      >D    ;
	      =     "MAL1S017Par".Par.FlagProcess1.FreshAirFlapCLOSE;

	      U     "MAL1S017Par".Par.FlagProcess1.FreshAirFlapOPEN;
	      U     "SYS_Scan0_Tick1min";
	      SPBN  dez;
	      L     "MAL1S017Par".Par.ParIntMachine.TargetPosWasteAir;
	      L     100; // limit max
	      >=I   ;
	      SPB   dez;
	      L     "MAL1S017Par".Par.ParIntMachine.TargetPosWasteAir;
	      L     1;
	      +I    ;
	      T     "MAL1S017Par".Par.ParIntMachine.TargetPosWasteAir;
	      SPA   e605;
	dez:  NOP   0;
	      U     "MAL1S017Par".Par.FlagProcess1.FreshAirFlapCLOSE;
	      U     "SYS_Scan0_Tick1min";
	      SPBN  e605;
	      L     "MAL1S017Par".Par.ParIntMachine.TargetPosWasteAir;
	      L     "MAL1S017Par".StepAct.PosFreshAirFlapBasic; // limit min
	      <=I   ;
	      SPB   e605;
	      L     "MAL1S017Par".Par.ParIntMachine.TargetPosWasteAir;
	      L     1;
	      -I    ;
	      T     "MAL1S017Par".Par.ParIntMachine.TargetPosWasteAir;
	      SPA   e605;

	summ: NOP   0;
	      L     "MAL1S017Par".StepAct.PosFreshAirFlapBasic;
	      T     "MAL1S017Par".Par.ParIntMachine.TargetPosWasteAir;
	      SPA   e605;

	e605: NOP   0;
	E605: NOP   0;
	NETWORK
	TITLE =ASW_6020: Copy germinating-recipe-data in Parameter DB
	      U     "MAL1S017Par".Par.FlagProcess.ProcessActive;
	      SPB   NoCl;
	// Clear process time in buffer
	      L     0;
	      T     "MAL1S017Par".ActTimeStepProcess.SteptimeActHour;
	      T     "MAL1S017Par".ActTimeStepProcess.SteptimeActMin;
	      T     "MAL1S017Par".ActTimeStepProcess.SteptimeActMinOverall;

	      T     "MAL1S017Par".Processtime.Day;
	      T     "MAL1S017Par".Processtime.Hour;
	      T     "MAL1S017Par".Processtime.Min;
	      T     "MAL1S017Par".Processtime.ProcessTimeActive;
	      L     L#0; // clear actual step time
	      T     "MAL1S017Par".Par.ProcessValue.StepTimeAct; // in ms

	NoCl: NOP   0;
	// Clear content recipe in buffer
	      L     0;
	      T     #tmpInt;
	      CALL "SIEMENS_FILL" (
		   BVAL                     := #tmpInt,
		   RET_VAL                  := #tmpRet,
		   BLK                      := "MAL1S017Par".RecipeHeader);
	//
	      U     "MAL1S017Par".Par.FlagFunction_1.StepUnloading;
	      UN    "MAL1S017Par".Par.FlagProcess.ProcessActive;
	      O     "MAL1S017Par".Par.FlagFunction_1.StepCleaning;
	      O     "MAL1S017Par".Par.FlagFunction_1.StepLoading;
	      SPBN  No00;
	// Germ: Copy step loading,unloading,cleaning to parameterDB
	      CALL "SIEMENS_BLKMOV" (
		   SRCBLK                   := "MAL1S017".SecNom.Germ.RecipeHeader.Loading,
		   RET_VAL                  := "MAL1S017Par".Par.Error.Value,
		   DSTBLK                   := "MAL1S017Par".RecipeHeader.Loading);
	      CALL "SIEMENS_BLKMOV" (
		   SRCBLK                   := "MAL1S017".SecNom.Germ.RecipeHeader.Unloading,
		   RET_VAL                  := "MAL1S017Par".Par.Error.Value,
		   DSTBLK                   := "MAL1S017Par".RecipeHeader.Unloading);
	      CALL "SIEMENS_BLKMOV" (
		   SRCBLK                   := "MAL1S017".SecNom.Germ.RecipeHeader.Cleaning,
		   RET_VAL                  := "MAL1S017Par".Par.Error.Value,
		   DSTBLK                   := "MAL1S017Par".RecipeHeader.Cleaning);

	No00: NOP   0;
	      U     "MAL1S017Par".Par.FlagProcess.ProcessActive;
	      SPBN  No03;
	// Germ: Copy common parameter
	      CALL "SIEMENS_BLKMOV" (
		   SRCBLK                   := "MAL1S017".SecNom.Germ.RecipeHeader,
		   RET_VAL                  := "MAL1S017Par".Par.Error.Value,
		   DSTBLK                   := "MAL1S017Par".RecipeHeader);
	//
	// Copy step parameter
	      U(    ;
	      L     "MAL1S017Par".Par.ParIntMachine.ActualStep;
	      L     1;
	      <I    ;
	      )     ;
	      O(    ;
	      L     "MAL1S017Par".Par.ParIntMachine.ActualStep;
	      L     "MAL1S017".SecNom.GERM.RecipeHeader.NumberOfSteps;
	      >I    ;
	      )     ;
	      SPB   NoXX; // error wrong step number
	      CALL "SYS_Copy_Array_Element" (
		   Source                   := "MAL1S017".SecNom.Germ.Step,
		   Destination              := "MAL1S017Par".StepAct,
		   Index                    := "MAL1S017Par".Par.ParIntMachine.ActualStep,
		   Fault                    := "MAL1S017Par".Par.Error.Bit);

	No03: NOP   0;
	NoXX: NOP   0;
	NETWORK
	TITLE =ASW_7000: Step loading germinating
	      U     "MAL1S017".ToASW.InfDataReady;
	      U     "MAL1S017".PCRead.Step.StWait;
	      U     "MAL1S017".PCWrite.ExtFuncOn.StartLoading; // PIC command "start loading"
	      S     "MAL1S017Par".Par.FlagFunction_1.StepLoading; // Step loading
	      SET;
	      R     "MAL1S017".PCWrite.ExtFuncOn.StartLoading; // PIC command "start loading"
	//

	      L     G100M.A_2111_MXZ41MA.Ma.OutPositionAngle;
	      L     3600; // 360,0°
	      >=I   ;
	      U     "MAL1S017".ToASW.InfDataReady;
	      U     "MAL1S017".PCRead.Step.StActive;
	      U     "MAL1S017Par".Par.FlagFunction_1.StepLoading; // Step loading
	      =     "MAL1S017Par".Par.FlagFunction_1.LoadFirstPartEnd;

	      U     "MAL1S017".ToASW.InfDataReady;
	      U     "MAL1S017".PCRead.Step.StActive;
	      U     "MAL1S017Par".Par.FlagFunction_1.StepLoading; // Step loading
	      SPBN  E700;
	      L     "MAL1S017Par".RecipeHeader.Loading.LiftingPositionRound_1;
	      T     "MAL1S017Par".Par.ParIntProcess.NextLevelLoading; // next level

	      U(    ;
	      L     G100M.A_2111_MXZ41MA.Ma.OutPositionAngle;
	      L     "MAL1S017Par".Par.ParIntProcess.NextLevelLoading; // next level
	      >=I   ;
	      )     ;
	      O     "MAL1S017Par".Par.FlagMachine_0.Speed2ndRound;
	      SPB   Rnd2;
	      L     "MAL1S017Par".RecipeHeader.Loading.LoadingLevelRound_1;
	      T     "MAL1S017Par".Par.MachineValue.SOLLWERT_HUBZUG1_HOEHE;
	      T     "MAL1S017Par".Par.MachineValue.SOLLWERT_HUBZUG2_HOEHE;

	      L     "MAL1S017Par".RecipeHeader.Loading.LoadingSpeed_1;
	      T     "MAL1S017Par".Par.MachineValue.SollwertFahrantrieb;

	      SPA   Rnd1;
	Rnd2: NOP   0;
	      L     "MAL1S017Par".RecipeHeader.Loading.LoadingLevelRound_2;
	      T     "MAL1S017Par".Par.MachineValue.SOLLWERT_HUBZUG1_HOEHE;
	      T     "MAL1S017Par".Par.MachineValue.SOLLWERT_HUBZUG2_HOEHE;
	      L     10;
	      T     WinCoS_BIW01_09PLC1BIW01_02.Ma.Par.ParTolPosition;

	      L     15; // 15Hz = Wendegeschwindigkeit
	      T     "MAL1S017Par".Par.MachineValue.SollwertFahrantrieb;

	// Sicherheitsbit; damit bei manueller Rückwärtsfahrt über die 346°-Marke, nicht mit Loading Speed_0 durch den gefüllten KK gefahren wird!!
	      SET   ;
	      S     "MAL1S017Par".Par.FlagMachine_0.Speed2ndRound;

	Rnd1: NOP   0;
	      U  M 50.0;
	      =  M 50.0;
	      L     "MAL1S017Par".Par.ParIntMachine.TargetPosTravDriveLoad; // 450 = endposition loading
	      T     G100M.A_2111_MXZ41MA.Ma.InPositionTarget;
	E700: NOP   0;
	NETWORK
	TITLE =Sub 7010: Germination loading finished
	//      U     "MAL1S017".ToASW.InfDataReady;
	//      U     "MAL1S017".PCRead.Step.StActive;
	//
	//      UN    "MAL1S017".ToASW.InfSameJobPrevSec;
	//      UN    "MAL1S017".PCRead.Step.StEmptying; // steep 1
	//      U     "MAL1S017".PCWrite.ExtFuncOn.FinishLoading; // PIC command "finish loading"
	//      U     "MAL1S017Par".Par.FlagFunction_1.StepLoading; // Step loading
	//      S     "MAL1S017Par".Par.FlagFunction_1.FinishLoading; // loading is finished start process germinating
	//      R     "MAL1S017Par".Par.FlagFunction_1.StepLoading; // Step loading
	//
	//      U     "MAL1S017".PCWrite.ExtFuncOn.FinishLoading; // PIC command "finish loading"
	//      R     "MAL1S017".PCWrite.ExtFuncOn.FinishLoading; // PIC command "finish loading"
	//
	//      U     "MAL1S017Par".Par.FlagFunction_1.StepLoading; // Step loading
	//      UN    "MAL1S017Par".Par.FlagFunction_1.FinishLoading; // loading is finished start process germinating
	//      SPBN  save;
	//      L     WinCoS_BIW01_09PLC1BIW01_02.Ma.OutPositionLeft;
	//      L     WinCoS_BIW01_09PLC1BIW01_02.Ma.OutPositionRight;
	//      +I    ;
	//      L     2;
	//      /I    ;
	//      T     "MAL1S017Par".Par.ParIntMachine.LastLoadingLevel; // saved loading value
	//save: NOP   0;
	//
	//      U     "MAL1S017".PCRead.Step.StReady;
	//      O     "MAL1S017".PCRead.Step.StActive;
	//      U     "MAL1S017Par".Par.FlagFunction_1.FinishLoading; // loading is finished start process germinating
	//      UN     "MAL1S017Par".Par.FlagFunction_1.StepLoading; // Step loading
	//      R     "MAL1S017Par".Par.FlagMachine_0.Speed2ndRound;
	//fin:  NOP   0;
	//E701: NOP   0;
	NETWORK
	TITLE =ASW_8000:  Step unloading germination
	        NOP 0;
	//      U     "MAL1S017".ToASW.InfDataReady
	//      U     "MAL1S017".PCRead.Step.StEmptying
	//      U     "MAL1S017".PCWrite.ExtFuncOn.StartUnLoading    // PIC command "start
	//      S     "MAL1S017Par".Par.FlagFunction_1.StepUnloading    // Step
	//      SET
	//      R     "MAL1S017".PCWrite.ExtFuncOn.StartUnLoading    // PIC command "start
	//
	      U  M 50.0;
	      =  M 50.0;
	      U     "MAL1S017".ToASW.InfDataReady;
	      U     "MAL1S017".PCRead.Step.StEmptying;
	      U     "MAL1S017".ToASW.InfSameJobNextSec;
	      UN    "MAL1S017Par".Par.FlagFunction_1.FinishUnloading;
	      =     "MAL1S017Par".Par.FlagFunction_1.StepUnloading; // Step Unloading
	//
	      U     "MAL1S017".ToASW.InfDataReady;
	      U     "MAL1S017".PCRead.Step.StEmptying;
	      U     "MAL1S017Par".Par.FlagFunction_1.StepUnloading; // Step Unloading
	      SPBN  e800;

	e800: NOP   0;
	M045: NOP   0;
	E800: NOP   0;
	NETWORK
	TITLE =ASW_9000: Step cleaning germination box
	      U     "MAL1S017".ToASW.InfDataReady;
	      U     "MAL1S017".PCRead.Step.StEmptied;
	      U     "MAL1S017Par".Par.FlagFunction_1.FinishUnloading;
	      U     "MAL1S017".PCWrite.ExtFuncOn.StartCleaning; // PIC command "start cleaning"
	      S     "MAL1S017Par".Par.FlagFunction_1.StepCleaning; // Step Cleaning
	      R     "MAL1S017Par".Par.FlagFunction_1.StepUnloading; // Step Unloading
	      SET;
	      R     "MAL1S017".PCWrite.ExtFuncOn.StartCleaning; // PIC command "start cleaning"

	      U     "MAL1S017".ToASW.InfDataReady;
	      U     "MAL1S017".PCRead.Step.StEmptied;
	      U     "MAL1S017Par".Par.FlagFunction_1.StepCleaning; // Step Cleaning
	      SPBN  e900;
	      L     3600; // 0°
	      T     G100M.A_2111_MXZ41MA.Ma.InPositionTarget;
	      U    M50.0;
	//    L     0
	//    T     G100M.A_2111_MXZ41MA.Ma.Par.ParTolPosition
	      =    M50.0;

	      L     "MAL1S017Par".RecipeHeader.Cleaning.CleaningSpeed_1;
	      T     "MAL1S017Par".Par.MachineValue.SollwertFahrantrieb;

	      L     "MAL1S017Par".RecipeHeader.Cleaning.CleaningLevel_1;
	      T     "MAL1S017Par".Par.MachineValue.SOLLWERT_HUBZUG1_HOEHE;
	      T     "MAL1S017Par".Par.MachineValue.SOLLWERT_HUBZUG2_HOEHE;

	      L     5;
	      T     WinCoS_BIW01_09PLC1BIW01_02.Ma.Par.ParTolPosition;
	e900: NOP   0;
	NETWORK
	TITLE =ASW_9010: Cleaning Germination box finished
	//
	      U     "MAL1S017".ToASW.InfDataReady;
	      U     "MAL1S017".PCRead.Step.StEmptied;
	      U     "MAL1S017Par".Par.FlagFunction_1.StepCleaning; // Step Cleaning
	      U     G100M.A_2111_MXZ41MA.Ma.OutAdjusted; // travelling drive on target position
	      U(;
	      U    M50.0;
	// Automaticly finishing cleaning
	      L     G100M.A_2111_MXZ41MA.IncCounter.VarInpHold;
	      L     L#12;                        // 8640[INK]/360°=24
	      <=D;
	      =    M50.0;
	// Command finishing cleaning
	      O     "MAL1S017".PCWrite.ExtFuncOn.FinishCleaning; // PIC command "cleaning finished"
	      );
	      S     "MAL1S017Par".Par.FlagFunction_1.FinishCleaning; // cleaning finished
	      R     "MAL1S017Par".Par.FlagFunction_1.StepCleaning; // Step Cleaning
	      R     "MAL1S017Par".Par.FlagFunction_1.FinishUnloading;

	      SET   ;
	      R     "MAL1S017".PCWrite.ExtFuncOn.FinishCleaning; // PIC command "cleaning finished"
	NETWORK
	TITLE =ASW_9080: Send section date to PIC after germination

	      AUF   "MAL1S017";
	      U     "MAL1S017".PCRead.Step.StEmptying;
	      FP    "MAL1S017Par".Par.FlagProcess.FP_SendResultToPIC;
	      SPBN  E908;
	//

	E908: NOP   0;
	NETWORK
	TITLE =ASW_10000: ILO functions
	//
	      U     "MAL1S017".SecAc.Sta1On.Inf08;
	      =     "MAL1S017".Gr.All.Spare04;

	//- Little help for PIC-People
	      U     "MAL1S017".SecAc.Sta1On.Inf08;
	      SPB   RSM;
	      L     0;
	      T     "MAL1S017Par".Ilo.Code_ILO_Funktion0; // FCM 17 LINE 1 SEC 17 GERM 1
	RSM:  NOP   0;

	//  no ILO-mode >> cmd manual off to all used groups and reset all flags
	      U     "MAL1S017".SecAc.Sta1On.Inf08;
	      FN    "MAL1S017Par".Ilo.Flag.EdgeILOModeOn;
	      S     "MAL1S017Par".Ilo.GrCMDManOff[1]; // (ManOff)
	      R     "MAL1S017Par".Ilo.GrCMDManAdditional.Cmd1[1];
	      R     "MAL1S017Par".Ilo.GrCMDManAdditional.Cmd2[2];
	//  Gr-cmd manual OFF
	      S     "G100M".Gr.CmdManualOff; // TRAVELLING DRIVE GERM 1
	      S     "G104M".Gr.CmdManualOff; // TURNING SCREWS GERM 1
	      S     "G105M".Gr.CmdManualOff; // FAN AND VALVE SRAY AIR GERM 1
	      S     "G106M".Gr.CmdManualOff; // FRESH AIR LOUVER GERM 1
	      S     "G107M".Gr.CmdManualOff; // EXHAUST AIR LOUVER GERM 1
	      S     "G112M".Gr.CmdManualOff; // COOLING / HEATING GERM 1
	//  RESET ADDITIONAL CMD`S
	      R     "G100M".USW14; // ILO-cmd
	      R     "G100M".USW15; // ILO-cmd
	      R     "G104M".USW14; // ILO-cmd
	      R     "G104M".USW15; // ILO-cmd
	      R     "G105M".USW14; // ILO-cmd
	      R     "G105M".USW15; // ILO-cmd
	      R     "G106M".USW14; // ILO-cmd
	      R     "G106M".USW15; // ILO-cmd
	      R     "G107M".USW14; // ILO-cmd
	      R     "G107M".USW15; // ILO-cmd
	      R     "G112M".USW14; // ILO-cmd
	      R     "G112M".USW15; // ILO-cmd
	//
	      NOP   0;
	// --- FCM 04 - Fans ---
	    L "MAL1S017Par".Ilo.ILOMode;
	    L  4;
	    <>I;
	    SPB IO4;
	// man on
	      U     "MAL1S017Par".Ilo.GrCMDManOn[1];
	      S     "G105M".Gr.InManual; // FAN AND VALVE SRAY AIR GERM 1
	      S     "G106M".Gr.InManual; // FRESH AIR LOUVER GERM 1
	      R     "MAL1S017Par".Ilo.GrCMDManOn[1];
	// man off
	      U     "MAL1S017Par".Ilo.GrCMDManOff[1];
	      S     "G105M".Gr.CmdManualOff; // FAN AND VALVE SRAY AIR GERM 1
	      R     "G105M".Gr.InManual; // FAN AND VALVE SRAY AIR GERM 1
	      R     "G105M".USW14; // ILO-cmd
	      R     "G105M".USW15; // ILO-cmd
	      S     "G106M".Gr.CmdManualOff; // FRESH AIR LOUVER GERM 1
	      R     "G106M".Gr.InManual; // FRESH AIR LOUVER GERM 1
	      R     "G106M".USW14; // ILO-cmd
	      R     "G106M".USW15; // ILO-cmd
	      R     "MAL1S017Par".Ilo.GrCMDManOff[1];
	      R     "MAL1S017Par".Ilo.GrCMDManAdditional.Cmd1[1];
	      R     "MAL1S017Par".Ilo.GrCMDManAdditional.Cmd2[1];
	// man start
	      U     "MAL1S017Par".Ilo.GrCMDManStart[1];
	      S     "G105M".Gr.CmdOn; // FAN AND VALVE SRAY AIR GERM 1
	      S     "G105M".Gr.CmdContinue; // FAN AND VALVE SRAY AIR GERM 1
	      S     "G106M".Gr.CmdOn; // FRESH AIR LOUVER GERM 1
	      S     "G106M".Gr.CmdContinue; // FRESH AIR LOUVER GERM 1
	      R     "MAL1S017Par".Ilo.GrCMDManStart[1];
	      U     "MAL1S017Par".Ilo.GrCMDManStart[2];
	      R     "MAL1S017Par".Ilo.GrCMDManStart[2];
	// man stop
	      U     "MAL1S017Par".Ilo.GrCMDManStop[1];
	      S     "G105M".Gr.CmdOff; // FAN AND VALVE SRAY AIR GERM 1
	      S     "G106M".Gr.CmdOff; // FRESH AIR LOUVER GERM 1
	      R     "MAL1S017Par".Ilo.GrCMDManStop[1];
	// man fault reset
	      U     "MAL1S017Par".Ilo.GrCMDManFaultReset[1];
	      S     "G105M".Gr.CmdFaultReset; // FAN AND VALVE SRAY AIR GERM 1
	      S     "G106M".Gr.CmdFaultReset; // FRESH AIR LOUVER GERM 1
	      R     "MAL1S017Par".Ilo.GrCMDManFaultReset[1];
	// target position
	      UN    "G105M".Gr.InManual; // FAN AND VALVE SRAY AIR GERM 1
	      O(;
	      L     "MAL1S017Par".Ilo.Code_ILO_Funktion0;
	      L     400;
	      <>I;
	      );
	      SPB   F04a;
	      L     "MAL1S017Par".Ilo.SetpointInt01[1];
	      T     "MAL1S017Par".Par.ParIntProcess.Speed_ILO_Fan;
	F04a:  NOP   0;

	IO4 : NOP   0;
	      NOP   0;
	// --- FCM 05 - Fans with target air temperature ---
	    L "MAL1S017Par".Ilo.ILOMode;
	    L  5;
	    <>I;
	    SPB IO5;
	// man on
	      U     "MAL1S017Par".Ilo.GrCMDManOn[1];
	      S     "G105M".Gr.InManual; // FAN AND VALVE SRAY AIR GERM 1
	      S     "G106M".Gr.InManual; // FRESH AIR LOUVER GERM 1
	      S     "G112M".Gr.InManual; // COOLING / HEATING GERM 1
	      R     "MAL1S017Par".Ilo.GrCMDManOn[1];
	// man off
	      U     "MAL1S017Par".Ilo.GrCMDManOff[1];
	      S     "G105M".Gr.CmdManualOff; // FAN AND VALVE SRAY AIR GERM 1
	      R     "G105M".Gr.InManual; // FAN AND VALVE SRAY AIR GERM 1
	      R     "G105M".USW14; // ILO-cmd
	      R     "G105M".USW15; // ILO-cmd
	      S     "G106M".Gr.CmdManualOff; // FRESH AIR LOUVER GERM 1
	      R     "G106M".Gr.InManual; // FRESH AIR LOUVER GERM 1
	      R     "G106M".USW14; // ILO-cmd
	      R     "G106M".USW15; // ILO-cmd
	      S     "G112M".Gr.CmdManualOff; // COOLING / HEATING GERM 1
	      R     "G112M".Gr.InManual; // COOLING / HEATING GERM 1
	      R     "G112M".USW14; // ILO-cmd
	      R     "G112M".USW15; // ILO-cmd
	      R     "MAL1S017Par".Ilo.GrCMDManOff[1];
	      R     "MAL1S017Par".Ilo.GrCMDManAdditional.Cmd1[1];
	      R     "MAL1S017Par".Ilo.GrCMDManAdditional.Cmd2[1];
	// man start
	      U     "MAL1S017Par".Ilo.GrCMDManStart[1];
	      S     "G105M".Gr.CmdOn; // FAN AND VALVE SRAY AIR GERM 1
	      S     "G105M".Gr.CmdContinue; // FAN AND VALVE SRAY AIR GERM 1
	      S     "G106M".Gr.CmdOn; // FRESH AIR LOUVER GERM 1
	      S     "G106M".Gr.CmdContinue; // FRESH AIR LOUVER GERM 1
	      S     "G112M".Gr.CmdOn; // COOLING / HEATING GERM 1
	      S     "G112M".Gr.CmdContinue; // COOLING / HEATING GERM 1
	      R     "MAL1S017Par".Ilo.GrCMDManStart[1];
	      U     "MAL1S017Par".Ilo.GrCMDManStart[2];
	      R     "MAL1S017Par".Ilo.GrCMDManStart[2];
	// man stop
	      U     "MAL1S017Par".Ilo.GrCMDManStop[1];
	      S     "G105M".Gr.CmdOff; // FAN AND VALVE SRAY AIR GERM 1
	      S     "G106M".Gr.CmdOff; // FRESH AIR LOUVER GERM 1
	      S     "G112M".Gr.CmdOff; // COOLING / HEATING GERM 1
	      R     "MAL1S017Par".Ilo.GrCMDManStop[1];
	// man fault reset
	      U     "MAL1S017Par".Ilo.GrCMDManFaultReset[1];
	      S     "G105M".Gr.CmdFaultReset; // FAN AND VALVE SRAY AIR GERM 1
	      S     "G106M".Gr.CmdFaultReset; // FRESH AIR LOUVER GERM 1
	      S     "G112M".Gr.CmdFaultReset; // COOLING / HEATING GERM 1
	      R     "MAL1S017Par".Ilo.GrCMDManFaultReset[1];
	// target position
	      UN    "G112M".Gr.InManual; // COOLING / HEATING GERM 1
	      SPB   F05a;
	      L     "MAL1S017Par".Ilo.SetpointInt02[1];    // Sollwert Temperatur
	      T     "MAL1S017Par".Par.ParIntProcess.TargetTemperature_ILO;
	F05a:  NOP   0;
	      UN    "G105M".Gr.InManual; // FAN AND VALVE SRAY AIR GERM 1
	      O(;
	      L     "MAL1S017Par".Ilo.Code_ILO_Funktion0;
	      L     500;
	      <>I;
	      );
	      SPB   F05b;
	      L     "MAL1S017Par".Ilo.SetpointInt01[1];
	      T     "MAL1S017Par".Par.ParIntProcess.Speed_ILO_Fan;
	F05b:  NOP   0;
	IO5 : NOP   0;
	      NOP   0;
	// --- FCM 06 - Fresh air flap ---
	    L "MAL1S017Par".Ilo.ILOMode;
	    L  6;
	    <>I;
	    SPB IO6;
	// man on
	      U     "MAL1S017Par".Ilo.GrCMDManOn[1];
	      S     "G106M".Gr.InManual; // FRESH AIR LOUVER GERM 1
	      R     "MAL1S017Par".Ilo.GrCMDManOn[1];
	// man off
	      U     "MAL1S017Par".Ilo.GrCMDManOff[1];
	      S     "G106M".Gr.CmdManualOff; // FRESH AIR LOUVER GERM 1
	      R     "G106M".Gr.InManual; // FRESH AIR LOUVER GERM 1
	      R     "G106M".USW14; // ILO-cmd
	      R     "G106M".USW15; // ILO-cmd
	      R     "MAL1S017Par".Ilo.GrCMDManOff[1];
	      R     "MAL1S017Par".Ilo.GrCMDManAdditional.Cmd1[1];
	      R     "MAL1S017Par".Ilo.GrCMDManAdditional.Cmd2[1];
	// man start
	      U     "MAL1S017Par".Ilo.GrCMDManStart[1];
	      S     "G106M".Gr.CmdOn; // FRESH AIR LOUVER GERM 1
	      S     "G106M".Gr.CmdContinue; // FRESH AIR LOUVER GERM 1
	      R     "MAL1S017Par".Ilo.GrCMDManStart[1];
	      U     "MAL1S017Par".Ilo.GrCMDManStart[2];
	      R     "MAL1S017Par".Ilo.GrCMDManStart[2];
	// man stop
	      U     "MAL1S017Par".Ilo.GrCMDManStop[1];
	      S     "G106M".Gr.CmdOff; // FRESH AIR LOUVER GERM 1
	      R     "MAL1S017Par".Ilo.GrCMDManStop[1];
	// man fault reset
	      U     "MAL1S017Par".Ilo.GrCMDManFaultReset[1];
	      S     "G106M".Gr.CmdFaultReset; // FRESH AIR LOUVER GERM 1
	      R     "MAL1S017Par".Ilo.GrCMDManFaultReset[1];
	// moving direction
	//
	// target position
	      UN    "G106M".Gr.InManual; // FRESH AIR LOUVER GERM 1
	      SPB   F06b;
	      L     "MAL1S017Par".Ilo.SetpointInt01[1];
	      T     "MAL1S017Par".Par.ParIntProcess.TarPos_ILO_FreshAir;
	F06b:  NOP   0;

	IO6 : NOP   0;
	      NOP   0;
	// --- FCM 09 - Floor drives ---
	    L "MAL1S017Par".Ilo.ILOMode;
	    L  9;
	    <>I;
	    SPB IO9;
	// man on
	      U     "MAL1S017Par".Ilo.GrCMDManOn[1];
	      S     "G100M".Gr.InManual; // TRAVELLING DRIVE GERM 1
	      S     "G104M".Gr.InManual; // TURNING SCREWS GERM 1
	      R     "MAL1S017Par".Ilo.GrCMDManOn[1];
	// man off
	      U     "MAL1S017Par".Ilo.GrCMDManOff[1];
	      S     "G100M".Gr.CmdManualOff; // TRAVELLING DRIVE GERM 1
	      R     "G100M".Gr.InManual; // TRAVELLING DRIVE GERM 1
	      R     "G100M".USW14; // ILO-cmd
	      R     "G100M".USW15; // ILO-cmd
	      S     "G104M".Gr.CmdManualOff; // TURNING SCREWS GERM 1
	      R     "G104M".Gr.InManual; // TURNING SCREWS GERM 1
	      R     "G104M".USW14; // ILO-cmd
	      R     "G104M".USW15; // ILO-cmd
	      R     "MAL1S017Par".Ilo.GrCMDManOff[1];
	      R     "MAL1S017Par".Ilo.GrCMDManAdditional.Cmd1[1];
	      R     "MAL1S017Par".Ilo.GrCMDManAdditional.Cmd2[1];
	// man start
	      U     "MAL1S017Par".Ilo.GrCMDManStart[1];
	      S     "G100M".Gr.CmdOn; // TRAVELLING DRIVE GERM 1
	      S     "G100M".Gr.CmdContinue; // TRAVELLING DRIVE GERM 1
	      S     "G104M".Gr.CmdOn; // TURNING SCREWS GERM 1
	      S     "G104M".Gr.CmdContinue; // TURNING SCREWS GERM 1
	      R     "MAL1S017Par".Ilo.GrCMDManStart[1];
	      U     "MAL1S017Par".Ilo.GrCMDManStart[2];
	      R     "MAL1S017Par".Ilo.GrCMDManStart[2];
	// man stop
	      U     "MAL1S017Par".Ilo.GrCMDManStop[1];
	      S     "G100M".Gr.CmdOff; // TRAVELLING DRIVE GERM 1
	      S     "G104M".Gr.CmdOff; // TURNING SCREWS GERM 1
	      R     "MAL1S017Par".Ilo.GrCMDManStop[1];
	// man fault reset
	      U     "MAL1S017Par".Ilo.GrCMDManFaultReset[1];
	      S     "G100M".Gr.CmdFaultReset; // TRAVELLING DRIVE GERM 1
	      S     "G104M".Gr.CmdFaultReset; // TURNING SCREWS GERM 1
	      R     "MAL1S017Par".Ilo.GrCMDManFaultReset[1];
	f091: NOP   0;
	      UN    "G100M".Gr.InManual; // TRAVELLING DRIVE GERM 1
	      O     ;
	      UN    "MAL1S017Par".Ilo.GrCMDManAdditional.Cmd1[1];
	      UN    "MAL1S017Par".Ilo.GrCMDManAdditional.Cmd2[1];
	      SPB   f092;
	      U     "MAL1S017Par".Ilo.GrCMDManAdditional.Cmd1[1];
	      =     "G100M".USW14; // ILO-cmd run fwd
	      U     "MAL1S017Par".Ilo.GrCMDManAdditional.Cmd2[1];
	      =     "G100M".USW15; // ILO-cmd run rev
	// target position
	      L     "MAL1S017Par".Ilo.SetpointInt01[1];
	      T     "MAL1S017Par".Par.ParIntProcess.Speed_ILO_FloorRotating;
	f092: NOP   0;

	IO9 : NOP   0;
	//
	// copy state
	      U     "G100M".Gr.InOutAutostartMan; // TRAVELLING DRIVE GERM 1
	      =     "MAL1S017Par".Ilo.GrSTMan[2];
	      U     "G104M".Gr.InOutAutostartMan; // TURNING SCREWS GERM 1
	      =     "MAL1S017Par".Ilo.GrSTMan[6];
	      U     "G105M".Gr.InOutAutostartMan; // FAN AND VALVE SRAY AIR GERM 1
	      =     "MAL1S017Par".Ilo.GrSTMan[7];
	      U     "G106M".Gr.InOutAutostartMan; // FRESH AIR LOUVER GERM 1
	      =     "MAL1S017Par".Ilo.GrSTMan[8];
	      U     "G107M".Gr.InOutAutostartMan; // EXHAUST AIR LOUVER GERM 1
	      =     "MAL1S017Par".Ilo.GrSTMan[9];
	      U     "G112M".Gr.InOutAutostartMan; // COOLING / HEATING GERM 1
	      =     "MAL1S017Par".Ilo.GrSTMan[14];
	NETWORK
	TITLE =ASW_9999: Init ASW Flags
	// clear all flags explicde to find them back
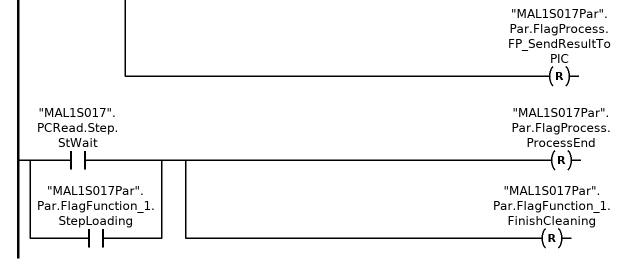
	      U     "MAL1S017".PCRead.Step.StPassive;
	      R     "MAL1S017Par".Par.FlagFunction_1.StepLoading;
	      R     "MAL1S017Par".Par.FlagFunction_1.StepUnloading;
	      R     "MAL1S017Par".Par.FlagFunction_1.StepCleaning;
	      R     "MAL1S017Par".Par.FlagFunction_1.LoadingBreak;
	      R     "MAL1S017Par".Par.FlagFunction_1.UnloadingBreak;
	      R     "MAL1S017Par".Par.FlagFunction_1.CleaningBreak;
	      R     "MAL1S017Par".Par.FlagFunction_1.FinishLoading;
	      R     "MAL1S017Par".Par.FlagFunction_1.FinishUnloading;
	      R     "MAL1S017Par".Par.FlagFunction_1.FinishCleaning;
	      R     "MAL1S017Par".Par.FlagFunction_1.Round_1;
	      R     "MAL1S017Par".Par.FlagFunction_1.Round_2;
	      R     "MAL1S017Par".Par.FlagFunction_1.Round_3;
	      R     "MAL1S017Par".Par.FlagFunction_1.Round_4;
	      R     "MAL1S017Par".Par.FlagFunction_1.Round_5;
	      R     "MAL1S017Par".Par.FlagFunction_1.Round_6;
	      R     "MAL1S017Par".Par.FlagFunction_1.Beladung_beendet;
	      R     "MAL1S017Par".Par.FlagFunction_1.Entladerunden_erreicht;
	      R     "MAL1S017Par".Par.FlagFunction_1.Reinigungsrunde_erreicht;
	      R     "MAL1S017Par".Par.FlagFunction_1.TurningStart;
	      R     "MAL1S017Par".Par.FlagFunction_1.TurningStop;
	      R     "MAL1S017Par".Par.FlagFunction_1.TurningLeft;
	      R     "MAL1S017Par".Par.FlagFunction_1.TurningRight;
	      R     "MAL1S017Par".Par.FlagFunction_1.LoadFirstPartEnd;
	      R     "MAL1S017Par".Par.FlagFunction_1.TurningWithSpraying;
	      R     "MAL1S017Par".Par.FlagFunction_1.TurningWithoutSpraying;
	      R     "MAL1S017Par".Par.FlagFunction_1.UnloadFirstPartEnd;
	      R     "MAL1S017Par".Par.FlagFunction_1.UnloadSecondPartEnd;
	      R     "MAL1S017Par".Par.FlagFunction_1.UnloadFirstPart;
	      R     "MAL1S017Par".Par.FlagFunction_1.UnloadSecondPart;
	      R     "MAL1S017Par".Par.FlagProcess.ProcessActive;
	      R     "MAL1S017Par".Par.FlagProcess.ProcessStartFP;
	      R     "MAL1S017Par".Par.FlagProcess.ProcessStartScan;
	      R     "MAL1S017Par".Par.FlagProcess.ProcessEnd;
	      R     "MAL1S017Par".Par.FlagProcess.FP_SendResultToPIC;
	      //
	      U     "MAL1S017".PCRead.Step.StWait;
	      O     "MAL1S017Par".Par.FlagFunction_1.StepLoading;
	      R     "MAL1S017Par".Par.FlagProcess.ProcessEnd;
	      R     "MAL1S017Par".Par.FlagFunction_1.FinishCleaning;

	NETWORK
	TITLE =Main0_End: Init flag
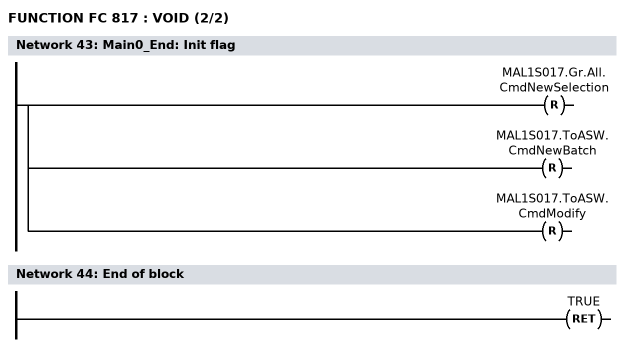
		SET;
		R     MAL1S017.Gr.All.CmdNewSelection;
		R     MAL1S017.ToASW.CmdNewBatch;
		R     MAL1S017.ToASW.CmdModify;

	NETWORK
	TITLE =End of block

	      BE    ;

	END_FUNCTION
